// TIA Portal V20 export
FUNCTION_BLOCK "Sequence_2_JROutPnPRight"   // FB32847, LAD
TITLE = Sequence
// Sequence template programmend in ladder logic
// stored: IsIECCheckEnabled true, MemoryReserve 100, Namespace Unit1.Em2, SetENOAutomatically true
   VAR_INPUT
      unitStatus : "LAF_typeUnitStatus";
   END_VAR
   VAR
      instSequenceLADControl { ExternalWritable := 'False'} : "LAF_ControlLadSequence";
      instSequenceLADStatus { ExternalWritable := 'False'} : "LAF_StatusLadSequence";
      statTonTime { ExternalWritable := 'False'} : Array[0..9999] of TON_TIME;
      NoDataCheck { S7_SetPoint := 'True'} : "LER_typePartData";
   END_VAR
   VAR_TEMP
      tempCustomerAction : Bool;   // Placeholder for possible actions
      tempDo_nothing_and_wait_for_init : Bool;   // Placeholder for doing nothing
      tempSafeStateCondition : Bool;   // Temp Condition for the equipment module to be in a safe state
   END_VAR
   VAR CONSTANT
      FALSE : Bool := FALSE;
      delayTime : Time := T#100ms;
      STEP_IDLE : DInt := 1;
      JOB_1_STEP_01 : DInt := 101;
      JOB_1_STEP_10 : DInt := 110;
      JOB_1_STEP_20 : DInt := 120;
      JOB_1_STEP_30 : DInt := 130;
      JOB_1_STEP_40 : DInt := 140;
      JOB_1_STEP_50 : DInt := 150;
      JOB_1_STEP_60 : DInt := 160;
      JOB_1_STEP_70 : DInt := 170;
      JOB_1_STEP_80 : DInt := 180;
      JOB_1_STEP_90 : DInt := 190;
      JOB_2_STEP_1 : DInt := 201;
      JOB_2_STEP_10 : DInt := 210;
      JOB_2_STEP_11 : DInt := 211;
      JOB_2_STEP_12 : DInt := 212;
      JOB_2_STEP_20 : DInt := 220;
      JOB_2_STEP_21 : DInt := 221;
      JOB_2_STEP_22 : DInt := 222;
      JOB_2_STEP_23 : DInt := 223;
      JOB_2_STEP_24 : DInt := 224;
      JOB_2_STEP_25 : DInt := 225;
      JOB_2_STEP_26 : DInt := 226;
      JOB_2_STEP_27 : DInt := 227;
      JOB_2_STEP_30 : DInt := 230;
      JOB_2_STEP_40 : DInt := 240;
      JOB_2_STEP_50 : DInt := 250;
      JOB_2_STEP_60 : DInt := 260;
      JOB_2_STEP_70 : DInt := 270;
      JOB_2_STEP_80 : DInt := 280;
      JOB_2_STEP_90 : DInt := 290;
      JOB_3_STEP_1 : DInt := 301;
      JOB_3_STEP_10 : DInt := 310;
      JOB_3_STEP_11 : DInt := 311;
      JOB_3_STEP_12 : DInt := 312;
      JOB_3_STEP_20 : DInt := 320;
      JOB_3_STEP_21 : DInt := 321;
      JOB_3_STEP_22 : DInt := 322;
      JOB_3_STEP_23 : DInt := 323;
      JOB_3_STEP_24 : DInt := 324;
      JOB_3_STEP_25 : DInt := 325;
      JOB_3_STEP_26 : DInt := 326;
      JOB_3_STEP_27 : DInt := 327;
      JOB_3_STEP_30 : DInt := 330;
      JOB_3_STEP_42 : DInt;
      JOB_3_STEP_31 : DInt := 331;
      JOB_3_STEP_40 : DInt := 340;
      JOB_3_STEP_41 : DInt := 341;
      JOB_3_STEP_50 : DInt := 350;
      JOB_3_STEP_51 : DInt := 351;
      JOB_3_STEP_60 : DInt := 360;
      JOB_3_STEP_70 : DInt := 370;
      JOB_3_STEP_80 : DInt := 380;
      JOB_3_STEP_90 : DInt := 390;
      STEP_IMMEDIATE_STOP : DInt := 9001;   // Step executed when an immediate stop command is triggered for the sequence (i.e. when unit is in state aborting)
      TO_DO_INSERT_ACTIONS_HERE : Bool := TRUE;   // Template : Add actions
      TO_DO_INSERT_CONDITION_FOR_TRANSITION_HERE : Bool := TRUE;   // Template : Add conditions
   END_VAR
   VAR_TEMP   // added for the SCL form of the ladder/FBD networks
      _w1 : Bool;
      _w2 : Bool;
      _w3 : Bool;
      _w4 : Bool;
      _w5 : Bool;
      _w6 : Bool;
      _w7 : Bool;
      _w8 : Bool;
   END_VAR
BEGIN

REGION Network 1: BLOCK INFO HEADER
   // (company) / (C) Copyright (year)
   // ---------------------------------------------------------------------------------
   // Title:                             (Title of this block)
   // Comment/Function: (that is implemented in the block)
   // Library/Family:           (that the source is dedicated to)
   // Author:                        (department / person in charge / contact)
   // Target System:          (test system with FW version)
   // Engineering:              TIA Portal (SW version)
   // Restrictions:               (OB types, etc.)
   // Requirements:           (hardware, technological package, etc.)
   // ---------------------------------------------------------------------------------
   // Change log table:
   // Version          | Date             | Signature      | Expert in charge  | Changes applied ------------------------|----------------------|-------------------------|--------------------------------|-----------------------
   // 001.000.000 | yyyy-mm-dd | 0x00000000 | (name of expert) | First released version
END_REGION

REGION Network 2: DESCRIPTION
   // This is a template block provided by the Automation Framework. It can be used to create an own project.
   // The Block Info Header is prepared to put in your own data.
   // Description of the block could be added here and the docu created by Code2Docu.
END_REGION

REGION Network 3: *************** CONTROL **********************
END_REGION

REGION Network 4: Sequence Control ("Enter your Sequins number here")
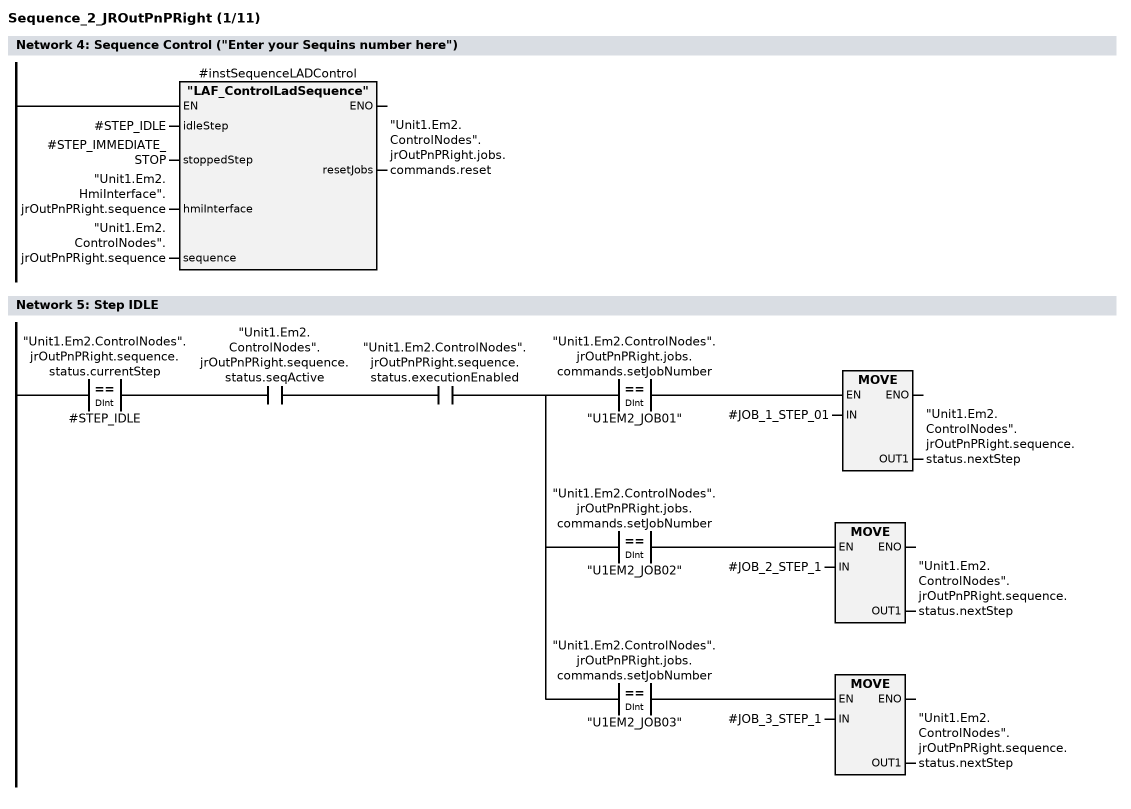
   RUNG wire#powerrail
      #instSequenceLADControl(idleStep := #STEP_IDLE, stoppedStep := #STEP_IMMEDIATE_STOP, hmiInterface := "Unit1.Em2.HmiInterface".jrOutPnPRight.sequence, sequence := "Unit1.Em2.ControlNodes".jrOutPnPRight.sequence, resetJobs => "Unit1.Em2.ControlNodes".jrOutPnPRight.jobs.commands.reset)
   END_RUNG
   // the same network as SCL:
   #instSequenceLADControl(idleStep := #STEP_IDLE,   // "LAF_ControlLadSequence"
                           stoppedStep := #STEP_IMMEDIATE_STOP,
                           hmiInterface := "Unit1.Em2.HmiInterface".jrOutPnPRight.sequence,
                           sequence := "Unit1.Em2.ControlNodes".jrOutPnPRight.sequence,
                           resetJobs => "Unit1.Em2.ControlNodes".jrOutPnPRight.jobs.commands.reset);
END_REGION

REGION Network 5: Step IDLE
   RUNG wire#powerrail
      { S7_Templates := "SrcType := DInt" } EQ_Contact(in1 := "Unit1.Em2.ControlNodes".jrOutPnPRight.sequence.status.currentStep, in2 := #STEP_IDLE)
      Contact( "Unit1.Em2.ControlNodes".jrOutPnPRight.sequence.status.seqActive )
      Contact( "Unit1.Em2.ControlNodes".jrOutPnPRight.sequence.status.executionEnabled )
      wire#w1
      { S7_Templates := "SrcType := DInt" } EQ_Contact(in1 := "Unit1.Em2.ControlNodes".jrOutPnPRight.jobs.commands.setJobNumber, in2 := "U1EM2_JOB01")
      Move(in := #JOB_1_STEP_01, out1 => "Unit1.Em2.ControlNodes".jrOutPnPRight.sequence.status.nextStep)
   END_RUNG
   RUNG wire#w1
      { S7_Templates := "SrcType := DInt" } EQ_Contact(in1 := "Unit1.Em2.ControlNodes".jrOutPnPRight.jobs.commands.setJobNumber, in2 := "U1EM2_JOB02")
      Move(in := #JOB_2_STEP_1, out1 => "Unit1.Em2.ControlNodes".jrOutPnPRight.sequence.status.nextStep)
   END_RUNG
   RUNG wire#w1
      { S7_Templates := "SrcType := DInt" } EQ_Contact(in1 := "Unit1.Em2.ControlNodes".jrOutPnPRight.jobs.commands.setJobNumber, in2 := "U1EM2_JOB03")
      Move(in := #JOB_3_STEP_1, out1 => "Unit1.Em2.ControlNodes".jrOutPnPRight.sequence.status.nextStep)
   END_RUNG
   // the same network as SCL:
   #_w1 := ("Unit1.Em2.ControlNodes".jrOutPnPRight.sequence.status.currentStep = #STEP_IDLE) AND "Unit1.Em2.ControlNodes".jrOutPnPRight.sequence.status.seqActive AND "Unit1.Em2.ControlNodes".jrOutPnPRight.sequence.status.executionEnabled;
   IF #_w1 AND ("Unit1.Em2.ControlNodes".jrOutPnPRight.jobs.commands.setJobNumber = "U1EM2_JOB01") THEN
       "Unit1.Em2.ControlNodes".jrOutPnPRight.sequence.status.nextStep := #JOB_1_STEP_01;
   END_IF;
   IF #_w1 AND ("Unit1.Em2.ControlNodes".jrOutPnPRight.jobs.commands.setJobNumber = "U1EM2_JOB02") THEN
       "Unit1.Em2.ControlNodes".jrOutPnPRight.sequence.status.nextStep := #JOB_2_STEP_1;
   END_IF;
   IF #_w1 AND ("Unit1.Em2.ControlNodes".jrOutPnPRight.jobs.commands.setJobNumber = "U1EM2_JOB03") THEN
       "Unit1.Em2.ControlNodes".jrOutPnPRight.sequence.status.nextStep := #JOB_3_STEP_1;
   END_IF;
END_REGION

REGION Network 6: *************** JOB[1] HOMING *************************
END_REGION

REGION Network 7: Step[101] : JOB[1] Condition
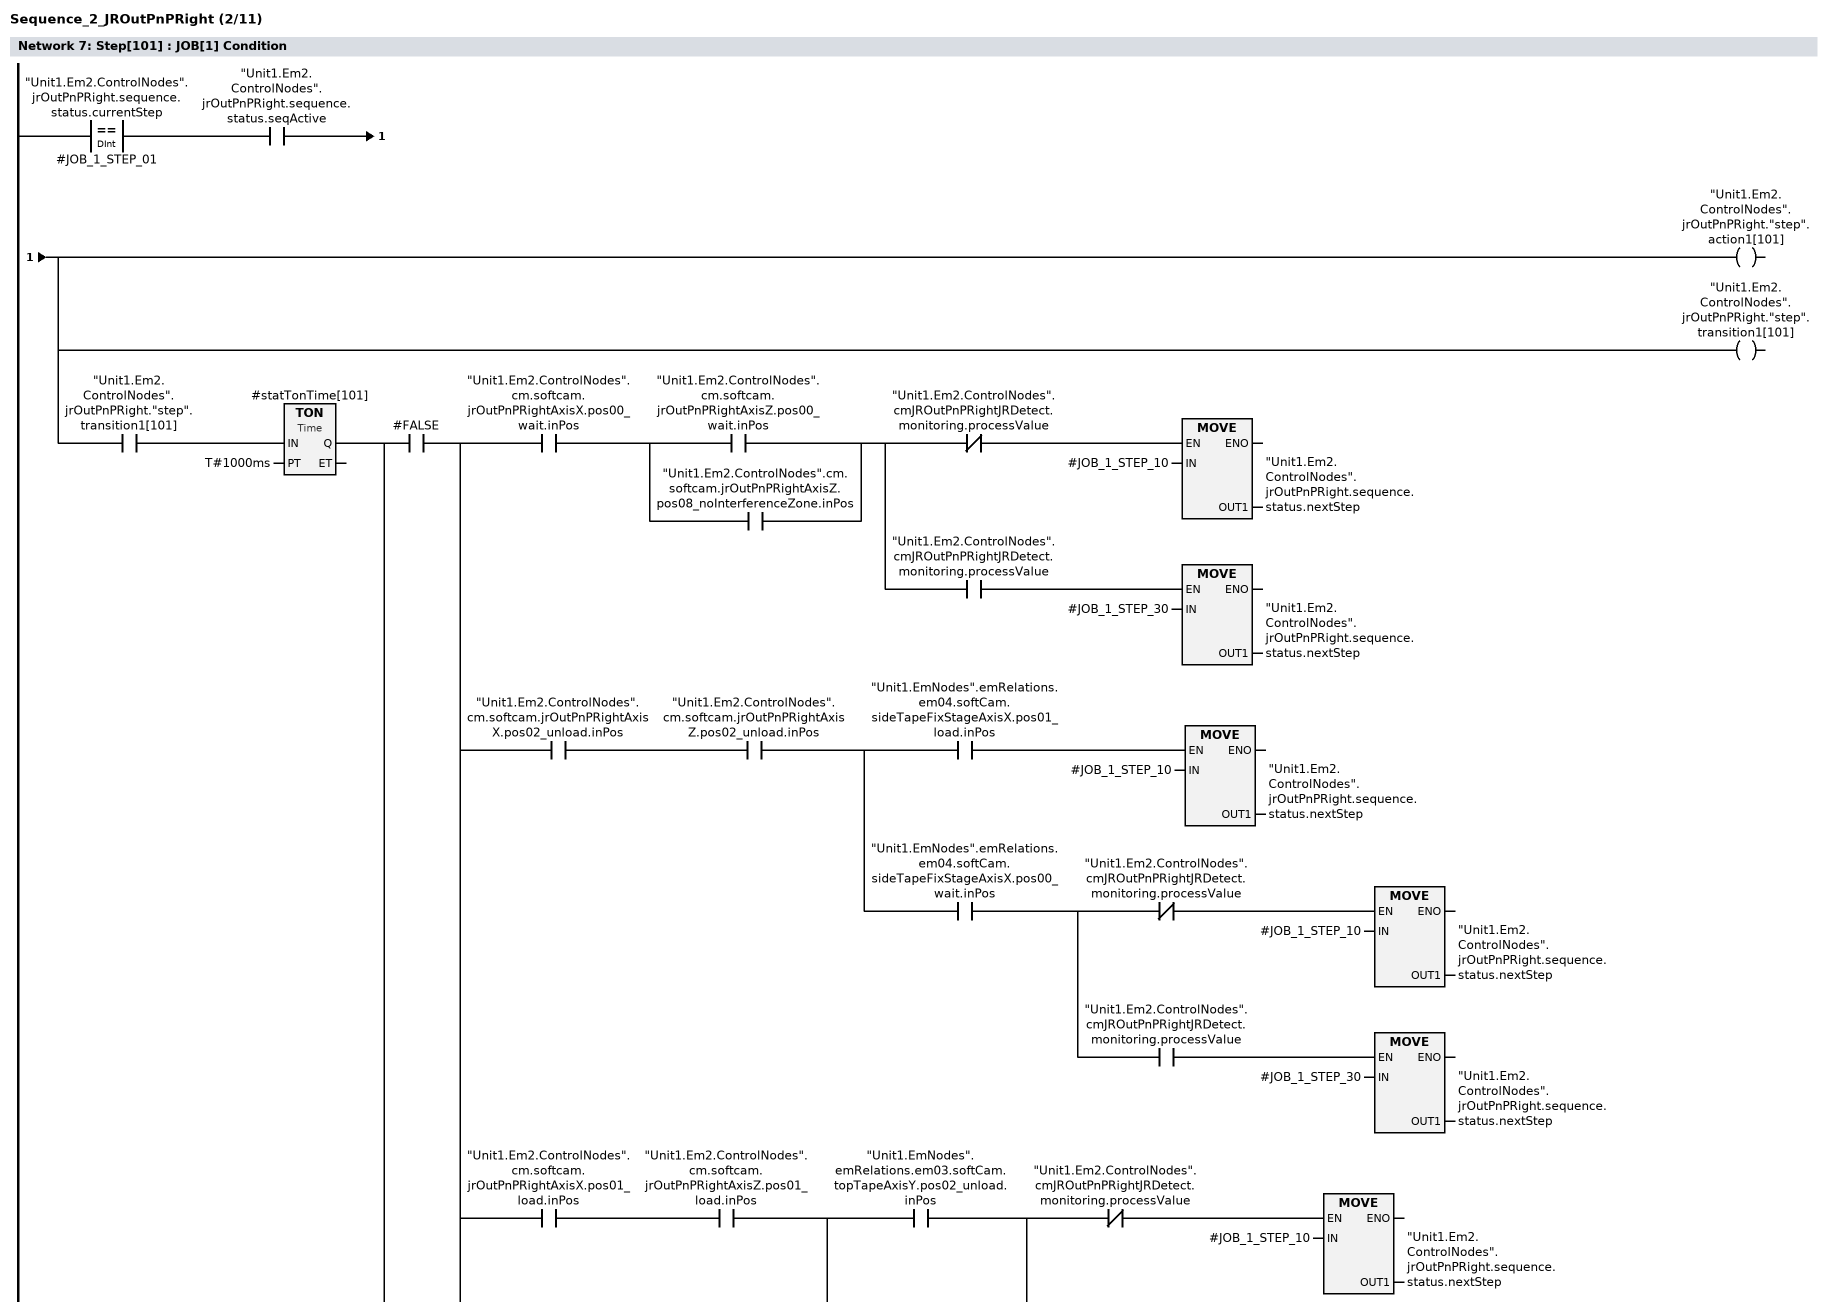
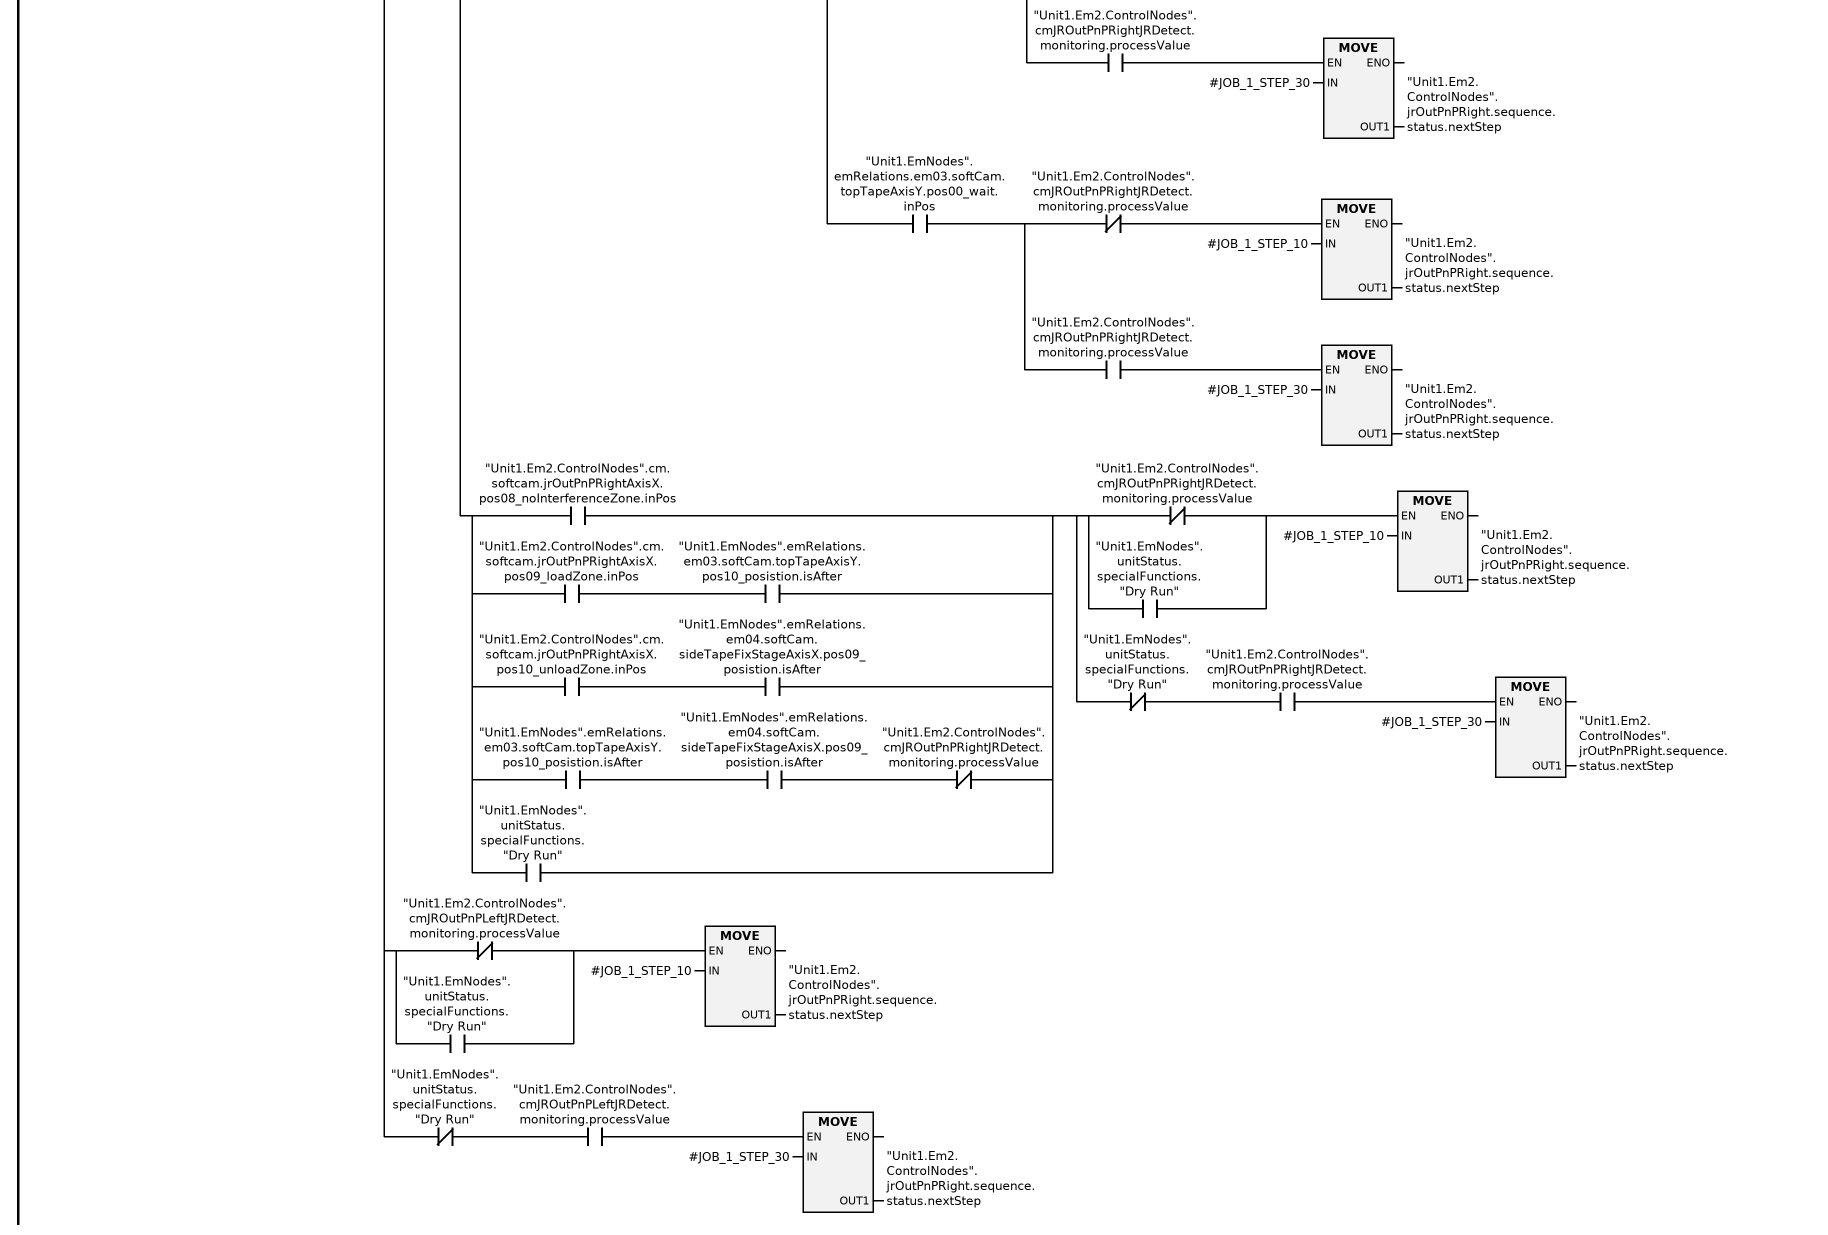
   RUNG wire#powerrail
      { S7_Templates := "SrcType := DInt" } EQ_Contact(in1 := "Unit1.Em2.ControlNodes".jrOutPnPRight.sequence.status.currentStep, in2 := #JOB_1_STEP_01)
      Contact( "Unit1.Em2.ControlNodes".jrOutPnPRight.sequence.status.seqActive )
      wire#w1
      Coil( "Unit1.Em2.ControlNodes".jrOutPnPRight."step".action1[101] )
   END_RUNG
   RUNG wire#w1
      Coil( "Unit1.Em2.ControlNodes".jrOutPnPRight."step".transition1[101] )
   END_RUNG
   RUNG wire#w1
      Contact( "Unit1.Em2.ControlNodes".jrOutPnPRight."step".transition1[101] )
      { S7_Templates := "time_type := Time" } #statTonTime[101].TON(pt := T#1000ms, et =>)
      wire#w2
      Contact( #FALSE )
      wire#w3
      Contact( "Unit1.Em2.ControlNodes".cm.softcam.jrOutPnPRightAxisX.pos00_wait.inPos )
      wire#w4
      Contact( "Unit1.Em2.ControlNodes".cm.softcam.jrOutPnPRightAxisZ.pos00_wait.inPos )
      wire#w5
      I_Contact( "Unit1.Em2.ControlNodes".cmJROutPnPRightJRDetect.monitoring.processValue )
      Move(in := #JOB_1_STEP_10, out1 => "Unit1.Em2.ControlNodes".jrOutPnPRight.sequence.status.nextStep)
   END_RUNG
   RUNG wire#w4
      Contact( "Unit1.Em2.ControlNodes".cm.softcam.jrOutPnPRightAxisZ.pos08_noInterferenceZone.inPos )
   END_RUNG wire#w5
   RUNG wire#w5
      Contact( "Unit1.Em2.ControlNodes".cmJROutPnPRightJRDetect.monitoring.processValue )
      Move(in := #JOB_1_STEP_30, out1 => "Unit1.Em2.ControlNodes".jrOutPnPRight.sequence.status.nextStep)
   END_RUNG
   RUNG wire#w3
      Contact( "Unit1.Em2.ControlNodes".cm.softcam.jrOutPnPRightAxisX.pos02_unload.inPos )
      Contact( "Unit1.Em2.ControlNodes".cm.softcam.jrOutPnPRightAxisZ.pos02_unload.inPos )
      wire#w6
      Contact( "Unit1.EmNodes".emRelations.em04.softCam.sideTapeFixStageAxisX.pos01_load.inPos )
      Move(in := #JOB_1_STEP_10, out1 => "Unit1.Em2.ControlNodes".jrOutPnPRight.sequence.status.nextStep)
   END_RUNG
   RUNG wire#w6
      Contact( "Unit1.EmNodes".emRelations.em04.softCam.sideTapeFixStageAxisX.pos00_wait.inPos )
      wire#w7
      I_Contact( "Unit1.Em2.ControlNodes".cmJROutPnPRightJRDetect.monitoring.processValue )
      Move(in := #JOB_1_STEP_10, out1 => "Unit1.Em2.ControlNodes".jrOutPnPRight.sequence.status.nextStep)
   END_RUNG
   RUNG wire#w7
      Contact( "Unit1.Em2.ControlNodes".cmJROutPnPRightJRDetect.monitoring.processValue )
      Move(in := #JOB_1_STEP_30, out1 => "Unit1.Em2.ControlNodes".jrOutPnPRight.sequence.status.nextStep)
   END_RUNG
   RUNG wire#w3
      Contact( "Unit1.Em2.ControlNodes".cm.softcam.jrOutPnPRightAxisX.pos01_load.inPos )
      Contact( "Unit1.Em2.ControlNodes".cm.softcam.jrOutPnPRightAxisZ.pos01_load.inPos )
      wire#w8
      Contact( "Unit1.EmNodes".emRelations.em03.softCam.topTapeAxisY.pos02_unload.inPos )
      wire#w9
      I_Contact( "Unit1.Em2.ControlNodes".cmJROutPnPRightJRDetect.monitoring.processValue )
      Move(in := #JOB_1_STEP_10, out1 => "Unit1.Em2.ControlNodes".jrOutPnPRight.sequence.status.nextStep)
   END_RUNG
   RUNG wire#w9
      Contact( "Unit1.Em2.ControlNodes".cmJROutPnPRightJRDetect.monitoring.processValue )
      Move(in := #JOB_1_STEP_30, out1 => "Unit1.Em2.ControlNodes".jrOutPnPRight.sequence.status.nextStep)
   END_RUNG
   RUNG wire#w8
      Contact( "Unit1.EmNodes".emRelations.em03.softCam.topTapeAxisY.pos00_wait.inPos )
      wire#w10
      I_Contact( "Unit1.Em2.ControlNodes".cmJROutPnPRightJRDetect.monitoring.processValue )
      Move(in := #JOB_1_STEP_10, out1 => "Unit1.Em2.ControlNodes".jrOutPnPRight.sequence.status.nextStep)
   END_RUNG
   RUNG wire#w10
      Contact( "Unit1.Em2.ControlNodes".cmJROutPnPRightJRDetect.monitoring.processValue )
      Move(in := #JOB_1_STEP_30, out1 => "Unit1.Em2.ControlNodes".jrOutPnPRight.sequence.status.nextStep)
   END_RUNG
   RUNG wire#w3
      Contact( "Unit1.Em2.ControlNodes".cm.softcam.jrOutPnPRightAxisX.pos08_noInterferenceZone.inPos )
      wire#w11
      I_Contact( "Unit1.Em2.ControlNodes".cmJROutPnPRightJRDetect.monitoring.processValue )
      wire#w12
      Move(in := #JOB_1_STEP_10, out1 => "Unit1.Em2.ControlNodes".jrOutPnPRight.sequence.status.nextStep)
   END_RUNG
   RUNG wire#w3
      Contact( "Unit1.Em2.ControlNodes".cm.softcam.jrOutPnPRightAxisX.pos09_loadZone.inPos )
      Contact( "Unit1.EmNodes".emRelations.em03.softCam.topTapeAxisY.pos10_posistion.isAfter )
   END_RUNG wire#w11
   RUNG wire#w3
      Contact( "Unit1.Em2.ControlNodes".cm.softcam.jrOutPnPRightAxisX.pos10_unloadZone.inPos )
      Contact( "Unit1.EmNodes".emRelations.em04.softCam.sideTapeFixStageAxisX.pos09_posistion.isAfter )
   END_RUNG wire#w11
   RUNG wire#w3
      Contact( "Unit1.EmNodes".emRelations.em03.softCam.topTapeAxisY.pos10_posistion.isAfter )
      Contact( "Unit1.EmNodes".emRelations.em04.softCam.sideTapeFixStageAxisX.pos09_posistion.isAfter )
      I_Contact( "Unit1.Em2.ControlNodes".cmJROutPnPRightJRDetect.monitoring.processValue )
   END_RUNG wire#w11
   RUNG wire#w3
      Contact( "Unit1.EmNodes".unitStatus.specialFunctions."Dry Run" )
   END_RUNG wire#w11
   RUNG wire#w11
      Contact( "Unit1.EmNodes".unitStatus.specialFunctions."Dry Run" )
   END_RUNG wire#w12
   RUNG wire#w11
      I_Contact( "Unit1.EmNodes".unitStatus.specialFunctions."Dry Run" )
      Contact( "Unit1.Em2.ControlNodes".cmJROutPnPRightJRDetect.monitoring.processValue )
      Move(in := #JOB_1_STEP_30, out1 => "Unit1.Em2.ControlNodes".jrOutPnPRight.sequence.status.nextStep)
   END_RUNG
   RUNG wire#w2
      I_Contact( "Unit1.Em2.ControlNodes".cmJROutPnPLeftJRDetect.monitoring.processValue )
      wire#w13
      Move(in := #JOB_1_STEP_10, out1 => "Unit1.Em2.ControlNodes".jrOutPnPRight.sequence.status.nextStep)
   END_RUNG
   RUNG wire#w2
      Contact( "Unit1.EmNodes".unitStatus.specialFunctions."Dry Run" )
   END_RUNG wire#w13
   RUNG wire#w2
      I_Contact( "Unit1.EmNodes".unitStatus.specialFunctions."Dry Run" )
      Contact( "Unit1.Em2.ControlNodes".cmJROutPnPLeftJRDetect.monitoring.processValue )
      Move(in := #JOB_1_STEP_30, out1 => "Unit1.Em2.ControlNodes".jrOutPnPRight.sequence.status.nextStep)
   END_RUNG
   // the same network as SCL:
   "Unit1.Em2.ControlNodes".jrOutPnPRight."step".action1[101] := ("Unit1.Em2.ControlNodes".jrOutPnPRight.sequence.status.currentStep = #JOB_1_STEP_01) AND "Unit1.Em2.ControlNodes".jrOutPnPRight.sequence.status.seqActive;
   "Unit1.Em2.ControlNodes".jrOutPnPRight."step".transition1[101] := ("Unit1.Em2.ControlNodes".jrOutPnPRight.sequence.status.currentStep = #JOB_1_STEP_01) AND "Unit1.Em2.ControlNodes".jrOutPnPRight.sequence.status.seqActive;
   #statTonTime[101].TON(IN := ("Unit1.Em2.ControlNodes".jrOutPnPRight.sequence.status.currentStep = #JOB_1_STEP_01) AND "Unit1.Em2.ControlNodes".jrOutPnPRight.sequence.status.seqActive AND "Unit1.Em2.ControlNodes".jrOutPnPRight."step".transition1[101],
                         PT := T#1000ms);
   #_w1 := #statTonTime[101].Q AND #FALSE;
   #_w2 := #_w1 AND "Unit1.Em2.ControlNodes".cm.softcam.jrOutPnPRightAxisX.pos00_wait.inPos AND ("Unit1.Em2.ControlNodes".cm.softcam.jrOutPnPRightAxisZ.pos00_wait.inPos OR "Unit1.Em2.ControlNodes".cm.softcam.jrOutPnPRightAxisZ.pos08_noInterferenceZone.inPos);
   IF #_w2 AND NOT "Unit1.Em2.ControlNodes".cmJROutPnPRightJRDetect.monitoring.processValue THEN
       "Unit1.Em2.ControlNodes".jrOutPnPRight.sequence.status.nextStep := #JOB_1_STEP_10;
   END_IF;
   IF #_w2 AND "Unit1.Em2.ControlNodes".cmJROutPnPRightJRDetect.monitoring.processValue THEN
       "Unit1.Em2.ControlNodes".jrOutPnPRight.sequence.status.nextStep := #JOB_1_STEP_30;
   END_IF;
   #_w3 := #_w1 AND "Unit1.Em2.ControlNodes".cm.softcam.jrOutPnPRightAxisX.pos02_unload.inPos AND "Unit1.Em2.ControlNodes".cm.softcam.jrOutPnPRightAxisZ.pos02_unload.inPos;
   IF #_w3 AND "Unit1.EmNodes".emRelations.em04.softCam.sideTapeFixStageAxisX.pos01_load.inPos THEN
       "Unit1.Em2.ControlNodes".jrOutPnPRight.sequence.status.nextStep := #JOB_1_STEP_10;
   END_IF;
   #_w4 := #_w3 AND "Unit1.EmNodes".emRelations.em04.softCam.sideTapeFixStageAxisX.pos00_wait.inPos;
   IF #_w4 AND NOT "Unit1.Em2.ControlNodes".cmJROutPnPRightJRDetect.monitoring.processValue THEN
       "Unit1.Em2.ControlNodes".jrOutPnPRight.sequence.status.nextStep := #JOB_1_STEP_10;
   END_IF;
   IF #_w4 AND "Unit1.Em2.ControlNodes".cmJROutPnPRightJRDetect.monitoring.processValue THEN
       "Unit1.Em2.ControlNodes".jrOutPnPRight.sequence.status.nextStep := #JOB_1_STEP_30;
   END_IF;
   #_w5 := #_w1 AND "Unit1.Em2.ControlNodes".cm.softcam.jrOutPnPRightAxisX.pos01_load.inPos AND "Unit1.Em2.ControlNodes".cm.softcam.jrOutPnPRightAxisZ.pos01_load.inPos;
   #_w6 := #_w5 AND "Unit1.EmNodes".emRelations.em03.softCam.topTapeAxisY.pos02_unload.inPos;
   IF #_w6 AND NOT "Unit1.Em2.ControlNodes".cmJROutPnPRightJRDetect.monitoring.processValue THEN
       "Unit1.Em2.ControlNodes".jrOutPnPRight.sequence.status.nextStep := #JOB_1_STEP_10;
   END_IF;
   IF #_w6 AND "Unit1.Em2.ControlNodes".cmJROutPnPRightJRDetect.monitoring.processValue THEN
       "Unit1.Em2.ControlNodes".jrOutPnPRight.sequence.status.nextStep := #JOB_1_STEP_30;
   END_IF;
   #_w7 := #_w5 AND "Unit1.EmNodes".emRelations.em03.softCam.topTapeAxisY.pos00_wait.inPos;
   IF #_w7 AND NOT "Unit1.Em2.ControlNodes".cmJROutPnPRightJRDetect.monitoring.processValue THEN
       "Unit1.Em2.ControlNodes".jrOutPnPRight.sequence.status.nextStep := #JOB_1_STEP_10;
   END_IF;
   IF #_w7 AND "Unit1.Em2.ControlNodes".cmJROutPnPRightJRDetect.monitoring.processValue THEN
       "Unit1.Em2.ControlNodes".jrOutPnPRight.sequence.status.nextStep := #JOB_1_STEP_30;
   END_IF;
   #_w8 := #_w1 AND ("Unit1.Em2.ControlNodes".cm.softcam.jrOutPnPRightAxisX.pos08_noInterferenceZone.inPos OR ("Unit1.Em2.ControlNodes".cm.softcam.jrOutPnPRightAxisX.pos09_loadZone.inPos AND "Unit1.EmNodes".emRelations.em03.softCam.topTapeAxisY.pos10_posistion.isAfter) OR ("Unit1.Em2.ControlNodes".cm.softcam.jrOutPnPRightAxisX.pos10_unloadZone.inPos AND "Unit1.EmNodes".emRelations.em04.softCam.sideTapeFixStageAxisX.pos09_posistion.isAfter) OR ("Unit1.EmNodes".emRelations.em03.softCam.topTapeAxisY.pos10_posistion.isAfter AND "Unit1.EmNodes".emRelations.em04.softCam.sideTapeFixStageAxisX.pos09_posistion.isAfter AND NOT "Unit1.Em2.ControlNodes".cmJROutPnPRightJRDetect.monitoring.processValue) OR "Unit1.EmNodes".unitStatus.specialFunctions."Dry Run");
   IF #_w8 AND (NOT "Unit1.Em2.ControlNodes".cmJROutPnPRightJRDetect.monitoring.processValue OR "Unit1.EmNodes".unitStatus.specialFunctions."Dry Run") THEN
       "Unit1.Em2.ControlNodes".jrOutPnPRight.sequence.status.nextStep := #JOB_1_STEP_10;
   END_IF;
   IF #_w8 AND NOT "Unit1.EmNodes".unitStatus.specialFunctions."Dry Run" AND "Unit1.Em2.ControlNodes".cmJROutPnPRightJRDetect.monitoring.processValue THEN
       "Unit1.Em2.ControlNodes".jrOutPnPRight.sequence.status.nextStep := #JOB_1_STEP_30;
   END_IF;
   IF #statTonTime[101].Q AND (NOT "Unit1.Em2.ControlNodes".cmJROutPnPLeftJRDetect.monitoring.processValue OR "Unit1.EmNodes".unitStatus.specialFunctions."Dry Run") THEN
       "Unit1.Em2.ControlNodes".jrOutPnPRight.sequence.status.nextStep := #JOB_1_STEP_10;
   END_IF;
   IF #statTonTime[101].Q AND NOT "Unit1.EmNodes".unitStatus.specialFunctions."Dry Run" AND "Unit1.Em2.ControlNodes".cmJROutPnPLeftJRDetect.monitoring.processValue THEN
       "Unit1.Em2.ControlNodes".jrOutPnPRight.sequence.status.nextStep := #JOB_1_STEP_30;
   END_IF;
END_REGION

REGION Network 8: Step[110] : JR PP Right Clamp Open
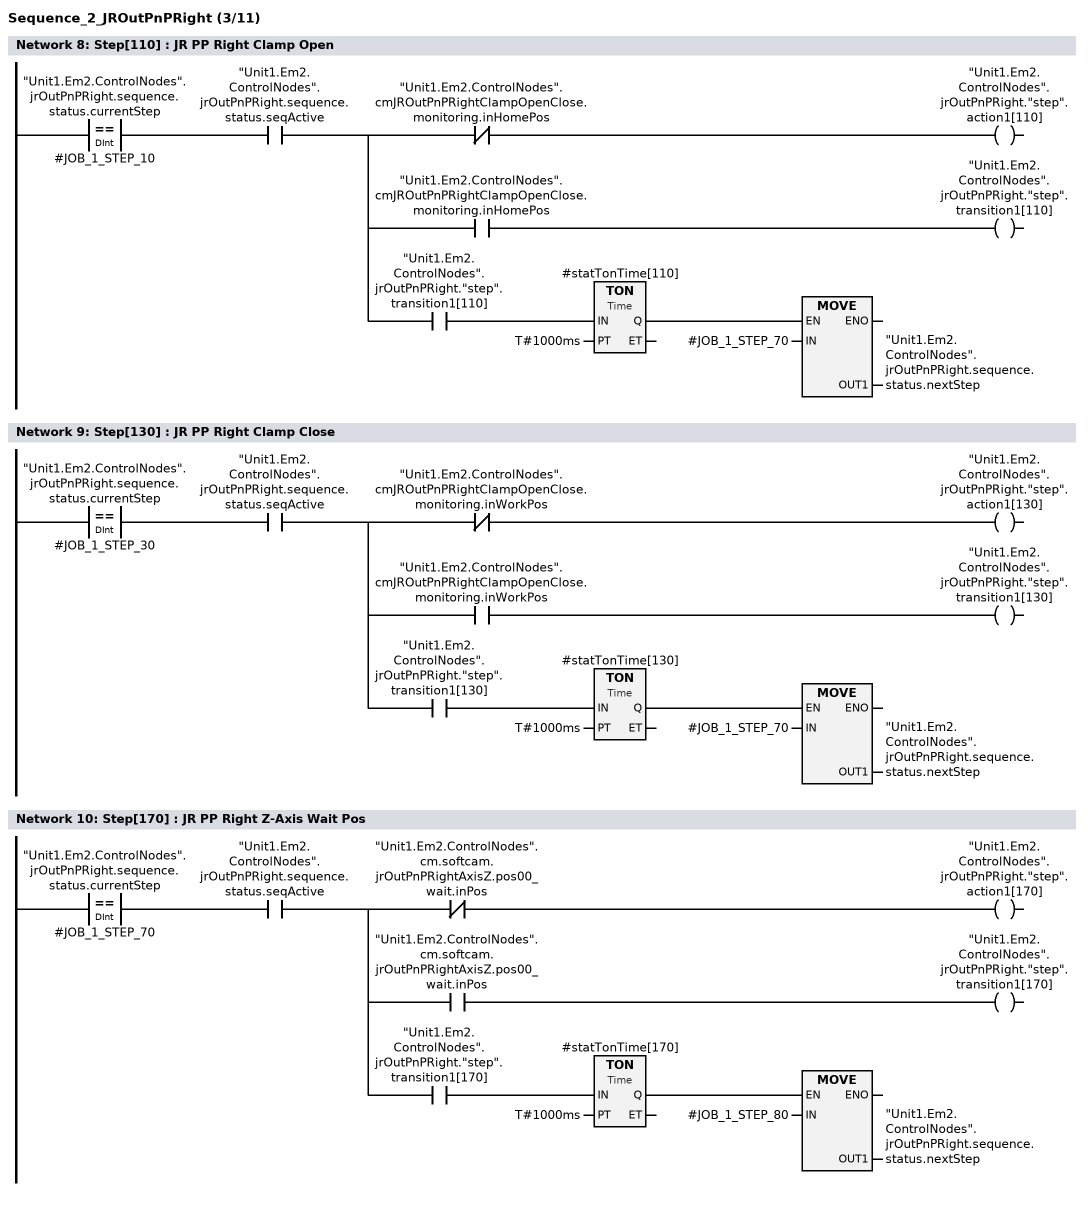
   RUNG wire#powerrail
      { S7_Templates := "SrcType := DInt" } EQ_Contact(in1 := "Unit1.Em2.ControlNodes".jrOutPnPRight.sequence.status.currentStep, in2 := #JOB_1_STEP_10)
      Contact( "Unit1.Em2.ControlNodes".jrOutPnPRight.sequence.status.seqActive )
      wire#w1
      I_Contact( "Unit1.Em2.ControlNodes".cmJROutPnPRightClampOpenClose.monitoring.inHomePos )
      Coil( "Unit1.Em2.ControlNodes".jrOutPnPRight."step".action1[110] )
   END_RUNG
   RUNG wire#w1
      Contact( "Unit1.Em2.ControlNodes".cmJROutPnPRightClampOpenClose.monitoring.inHomePos )
      Coil( "Unit1.Em2.ControlNodes".jrOutPnPRight."step".transition1[110] )
   END_RUNG
   RUNG wire#w1
      Contact( "Unit1.Em2.ControlNodes".jrOutPnPRight."step".transition1[110] )
      { S7_Templates := "time_type := Time" } #statTonTime[110].TON(pt := T#1000ms, et =>)
      Move(in := #JOB_1_STEP_70, out1 => "Unit1.Em2.ControlNodes".jrOutPnPRight.sequence.status.nextStep)
   END_RUNG
   // the same network as SCL:
   #_w1 := ("Unit1.Em2.ControlNodes".jrOutPnPRight.sequence.status.currentStep = #JOB_1_STEP_10) AND "Unit1.Em2.ControlNodes".jrOutPnPRight.sequence.status.seqActive;
   "Unit1.Em2.ControlNodes".jrOutPnPRight."step".action1[110] := #_w1 AND NOT "Unit1.Em2.ControlNodes".cmJROutPnPRightClampOpenClose.monitoring.inHomePos;
   "Unit1.Em2.ControlNodes".jrOutPnPRight."step".transition1[110] := #_w1 AND "Unit1.Em2.ControlNodes".cmJROutPnPRightClampOpenClose.monitoring.inHomePos;
   #statTonTime[110].TON(IN := #_w1 AND "Unit1.Em2.ControlNodes".jrOutPnPRight."step".transition1[110],
                         PT := T#1000ms);
   IF #statTonTime[110].Q THEN
       "Unit1.Em2.ControlNodes".jrOutPnPRight.sequence.status.nextStep := #JOB_1_STEP_70;
   END_IF;
END_REGION

REGION Network 9: Step[130] : JR PP Right Clamp Close
   RUNG wire#powerrail
      { S7_Templates := "SrcType := DInt" } EQ_Contact(in1 := "Unit1.Em2.ControlNodes".jrOutPnPRight.sequence.status.currentStep, in2 := #JOB_1_STEP_30)
      Contact( "Unit1.Em2.ControlNodes".jrOutPnPRight.sequence.status.seqActive )
      wire#w1
      I_Contact( "Unit1.Em2.ControlNodes".cmJROutPnPRightClampOpenClose.monitoring.inWorkPos )
      Coil( "Unit1.Em2.ControlNodes".jrOutPnPRight."step".action1[130] )
   END_RUNG
   RUNG wire#w1
      Contact( "Unit1.Em2.ControlNodes".cmJROutPnPRightClampOpenClose.monitoring.inWorkPos )
      Coil( "Unit1.Em2.ControlNodes".jrOutPnPRight."step".transition1[130] )
   END_RUNG
   RUNG wire#w1
      Contact( "Unit1.Em2.ControlNodes".jrOutPnPRight."step".transition1[130] )
      { S7_Templates := "time_type := Time" } #statTonTime[130].TON(pt := T#1000ms, et =>)
      Move(in := #JOB_1_STEP_70, out1 => "Unit1.Em2.ControlNodes".jrOutPnPRight.sequence.status.nextStep)
   END_RUNG
   // the same network as SCL:
   #_w1 := ("Unit1.Em2.ControlNodes".jrOutPnPRight.sequence.status.currentStep = #JOB_1_STEP_30) AND "Unit1.Em2.ControlNodes".jrOutPnPRight.sequence.status.seqActive;
   "Unit1.Em2.ControlNodes".jrOutPnPRight."step".action1[130] := #_w1 AND NOT "Unit1.Em2.ControlNodes".cmJROutPnPRightClampOpenClose.monitoring.inWorkPos;
   "Unit1.Em2.ControlNodes".jrOutPnPRight."step".transition1[130] := #_w1 AND "Unit1.Em2.ControlNodes".cmJROutPnPRightClampOpenClose.monitoring.inWorkPos;
   #statTonTime[130].TON(IN := #_w1 AND "Unit1.Em2.ControlNodes".jrOutPnPRight."step".transition1[130],
                         PT := T#1000ms);
   IF #statTonTime[130].Q THEN
       "Unit1.Em2.ControlNodes".jrOutPnPRight.sequence.status.nextStep := #JOB_1_STEP_70;
   END_IF;
END_REGION

REGION Network 10: Step[170] : JR PP Right Z-Axis Wait Pos
   RUNG wire#powerrail
      { S7_Templates := "SrcType := DInt" } EQ_Contact(in1 := "Unit1.Em2.ControlNodes".jrOutPnPRight.sequence.status.currentStep, in2 := #JOB_1_STEP_70)
      Contact( "Unit1.Em2.ControlNodes".jrOutPnPRight.sequence.status.seqActive )
      wire#w1
      I_Contact( "Unit1.Em2.ControlNodes".cm.softcam.jrOutPnPRightAxisZ.pos00_wait.inPos )
      Coil( "Unit1.Em2.ControlNodes".jrOutPnPRight."step".action1[170] )
   END_RUNG
   RUNG wire#w1
      Contact( "Unit1.Em2.ControlNodes".cm.softcam.jrOutPnPRightAxisZ.pos00_wait.inPos )
      Coil( "Unit1.Em2.ControlNodes".jrOutPnPRight."step".transition1[170] )
   END_RUNG
   RUNG wire#w1
      Contact( "Unit1.Em2.ControlNodes".jrOutPnPRight."step".transition1[170] )
      { S7_Templates := "time_type := Time" } #statTonTime[170].TON(pt := T#1000ms, et =>)
      Move(in := #JOB_1_STEP_80, out1 => "Unit1.Em2.ControlNodes".jrOutPnPRight.sequence.status.nextStep)
   END_RUNG
   // the same network as SCL:
   #_w1 := ("Unit1.Em2.ControlNodes".jrOutPnPRight.sequence.status.currentStep = #JOB_1_STEP_70) AND "Unit1.Em2.ControlNodes".jrOutPnPRight.sequence.status.seqActive;
   "Unit1.Em2.ControlNodes".jrOutPnPRight."step".action1[170] := #_w1 AND NOT "Unit1.Em2.ControlNodes".cm.softcam.jrOutPnPRightAxisZ.pos00_wait.inPos;
   "Unit1.Em2.ControlNodes".jrOutPnPRight."step".transition1[170] := #_w1 AND "Unit1.Em2.ControlNodes".cm.softcam.jrOutPnPRightAxisZ.pos00_wait.inPos;
   #statTonTime[170].TON(IN := #_w1 AND "Unit1.Em2.ControlNodes".jrOutPnPRight."step".transition1[170],
                         PT := T#1000ms);
   IF #statTonTime[170].Q THEN
       "Unit1.Em2.ControlNodes".jrOutPnPRight.sequence.status.nextStep := #JOB_1_STEP_80;
   END_IF;
END_REGION

REGION Network 11: Step[180] : JR PP Right X-Axis Wait Pos
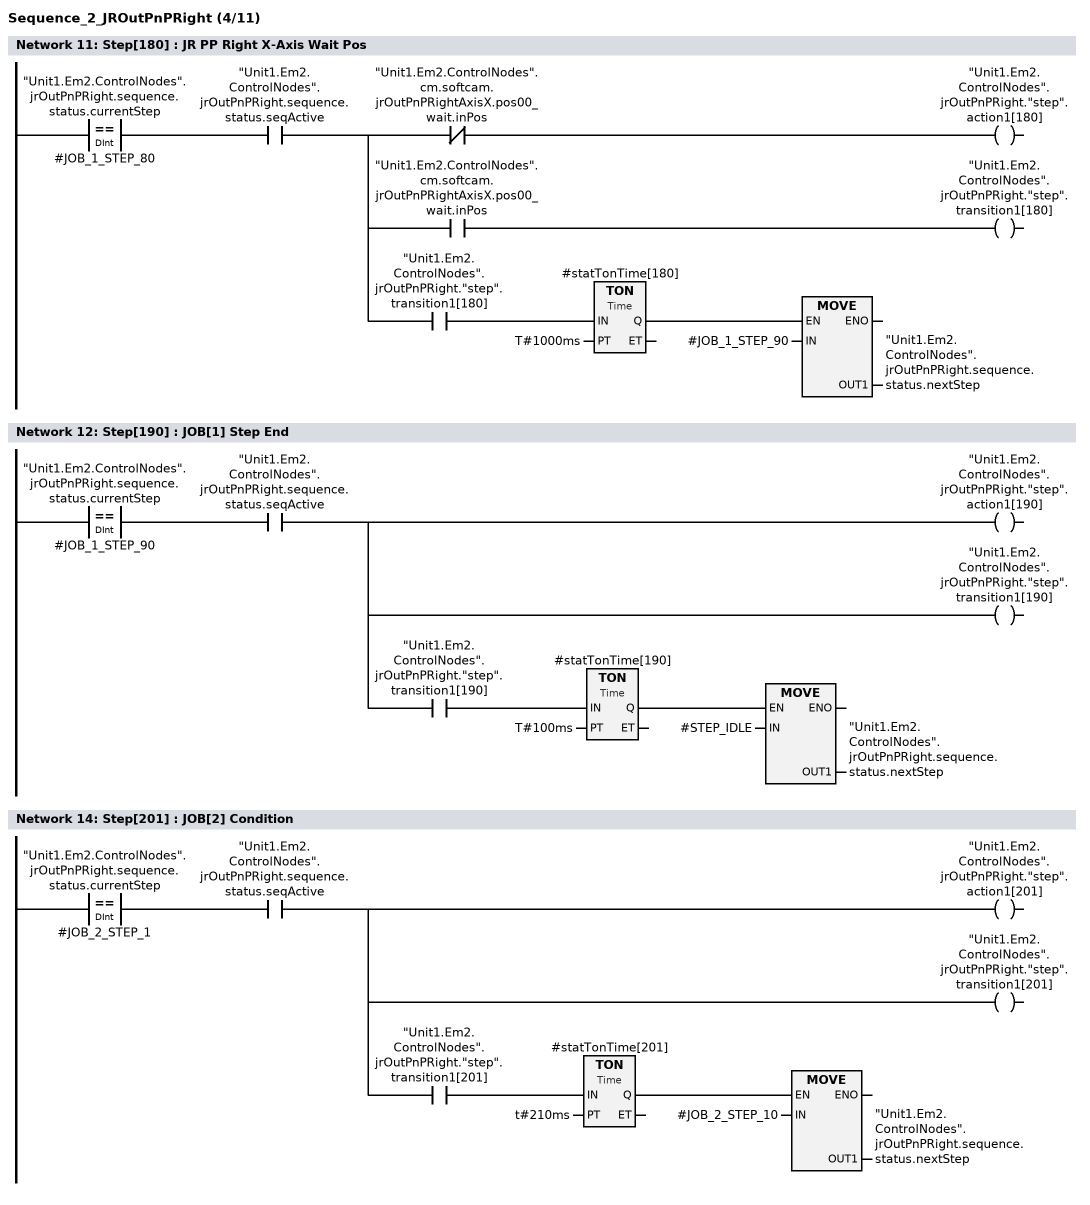
   RUNG wire#powerrail
      { S7_Templates := "SrcType := DInt" } EQ_Contact(in1 := "Unit1.Em2.ControlNodes".jrOutPnPRight.sequence.status.currentStep, in2 := #JOB_1_STEP_80)
      Contact( "Unit1.Em2.ControlNodes".jrOutPnPRight.sequence.status.seqActive )
      wire#w1
      I_Contact( "Unit1.Em2.ControlNodes".cm.softcam.jrOutPnPRightAxisX.pos00_wait.inPos )
      Coil( "Unit1.Em2.ControlNodes".jrOutPnPRight."step".action1[180] )
   END_RUNG
   RUNG wire#w1
      Contact( "Unit1.Em2.ControlNodes".cm.softcam.jrOutPnPRightAxisX.pos00_wait.inPos )
      Coil( "Unit1.Em2.ControlNodes".jrOutPnPRight."step".transition1[180] )
   END_RUNG
   RUNG wire#w1
      Contact( "Unit1.Em2.ControlNodes".jrOutPnPRight."step".transition1[180] )
      { S7_Templates := "time_type := Time" } #statTonTime[180].TON(pt := T#1000ms, et =>)
      Move(in := #JOB_1_STEP_90, out1 => "Unit1.Em2.ControlNodes".jrOutPnPRight.sequence.status.nextStep)
   END_RUNG
   // the same network as SCL:
   #_w1 := ("Unit1.Em2.ControlNodes".jrOutPnPRight.sequence.status.currentStep = #JOB_1_STEP_80) AND "Unit1.Em2.ControlNodes".jrOutPnPRight.sequence.status.seqActive;
   "Unit1.Em2.ControlNodes".jrOutPnPRight."step".action1[180] := #_w1 AND NOT "Unit1.Em2.ControlNodes".cm.softcam.jrOutPnPRightAxisX.pos00_wait.inPos;
   "Unit1.Em2.ControlNodes".jrOutPnPRight."step".transition1[180] := #_w1 AND "Unit1.Em2.ControlNodes".cm.softcam.jrOutPnPRightAxisX.pos00_wait.inPos;
   #statTonTime[180].TON(IN := #_w1 AND "Unit1.Em2.ControlNodes".jrOutPnPRight."step".transition1[180],
                         PT := T#1000ms);
   IF #statTonTime[180].Q THEN
       "Unit1.Em2.ControlNodes".jrOutPnPRight.sequence.status.nextStep := #JOB_1_STEP_90;
   END_IF;
END_REGION

REGION Network 12: Step[190] : JOB[1] Step End
   RUNG wire#powerrail
      { S7_Templates := "SrcType := DInt" } EQ_Contact(in1 := "Unit1.Em2.ControlNodes".jrOutPnPRight.sequence.status.currentStep, in2 := #JOB_1_STEP_90)
      Contact( "Unit1.Em2.ControlNodes".jrOutPnPRight.sequence.status.seqActive )
      wire#w1
      Coil( "Unit1.Em2.ControlNodes".jrOutPnPRight."step".action1[190] )
   END_RUNG
   RUNG wire#w1
      Coil( "Unit1.Em2.ControlNodes".jrOutPnPRight."step".transition1[190] )
   END_RUNG
   RUNG wire#w1
      Contact( "Unit1.Em2.ControlNodes".jrOutPnPRight."step".transition1[190] )
      { S7_Templates := "time_type := Time" } #statTonTime[190].TON(pt := T#100ms, et =>)
      Move(in := #STEP_IDLE, out1 => "Unit1.Em2.ControlNodes".jrOutPnPRight.sequence.status.nextStep)
   END_RUNG
   // the same network as SCL:
   "Unit1.Em2.ControlNodes".jrOutPnPRight."step".action1[190] := ("Unit1.Em2.ControlNodes".jrOutPnPRight.sequence.status.currentStep = #JOB_1_STEP_90) AND "Unit1.Em2.ControlNodes".jrOutPnPRight.sequence.status.seqActive;
   "Unit1.Em2.ControlNodes".jrOutPnPRight."step".transition1[190] := ("Unit1.Em2.ControlNodes".jrOutPnPRight.sequence.status.currentStep = #JOB_1_STEP_90) AND "Unit1.Em2.ControlNodes".jrOutPnPRight.sequence.status.seqActive;
   #statTonTime[190].TON(IN := ("Unit1.Em2.ControlNodes".jrOutPnPRight.sequence.status.currentStep = #JOB_1_STEP_90) AND "Unit1.Em2.ControlNodes".jrOutPnPRight.sequence.status.seqActive AND "Unit1.Em2.ControlNodes".jrOutPnPRight."step".transition1[190],
                         PT := T#100ms);
   IF #statTonTime[190].Q THEN
       "Unit1.Em2.ControlNodes".jrOutPnPRight.sequence.status.nextStep := #STEP_IDLE;
   END_IF;
END_REGION

REGION Network 13: *************** JOB[2] JR GET TOP TAPE FIX STAGE=AUTO *************************
END_REGION

REGION Network 14: Step[201] : JOB[2] Condition
   RUNG wire#powerrail
      { S7_Templates := "SrcType := DInt" } EQ_Contact(in1 := "Unit1.Em2.ControlNodes".jrOutPnPRight.sequence.status.currentStep, in2 := #JOB_2_STEP_1)
      Contact( "Unit1.Em2.ControlNodes".jrOutPnPRight.sequence.status.seqActive )
      wire#w1
      Coil( "Unit1.Em2.ControlNodes".jrOutPnPRight."step".action1[201] )
   END_RUNG
   RUNG wire#w1
      Coil( "Unit1.Em2.ControlNodes".jrOutPnPRight."step".transition1[201] )
   END_RUNG
   RUNG wire#w1
      Contact( "Unit1.Em2.ControlNodes".jrOutPnPRight."step".transition1[201] )
      { S7_Templates := "time_type := Time" } #statTonTime[201].TON(pt := t#210ms, et =>)
      Move(in := #JOB_2_STEP_10, out1 => "Unit1.Em2.ControlNodes".jrOutPnPRight.sequence.status.nextStep)
   END_RUNG
   // the same network as SCL:
   "Unit1.Em2.ControlNodes".jrOutPnPRight."step".action1[201] := ("Unit1.Em2.ControlNodes".jrOutPnPRight.sequence.status.currentStep = #JOB_2_STEP_1) AND "Unit1.Em2.ControlNodes".jrOutPnPRight.sequence.status.seqActive;
   "Unit1.Em2.ControlNodes".jrOutPnPRight."step".transition1[201] := ("Unit1.Em2.ControlNodes".jrOutPnPRight.sequence.status.currentStep = #JOB_2_STEP_1) AND "Unit1.Em2.ControlNodes".jrOutPnPRight.sequence.status.seqActive;
   #statTonTime[201].TON(IN := ("Unit1.Em2.ControlNodes".jrOutPnPRight.sequence.status.currentStep = #JOB_2_STEP_1) AND "Unit1.Em2.ControlNodes".jrOutPnPRight.sequence.status.seqActive AND "Unit1.Em2.ControlNodes".jrOutPnPRight."step".transition1[201],
                         PT := t#210ms);
   IF #statTonTime[201].Q THEN
       "Unit1.Em2.ControlNodes".jrOutPnPRight.sequence.status.nextStep := #JOB_2_STEP_10;
   END_IF;
END_REGION

REGION Network 15: Step[210] : JR PP Right X-Axis Loading Pos[Top Tape Fix Stage]
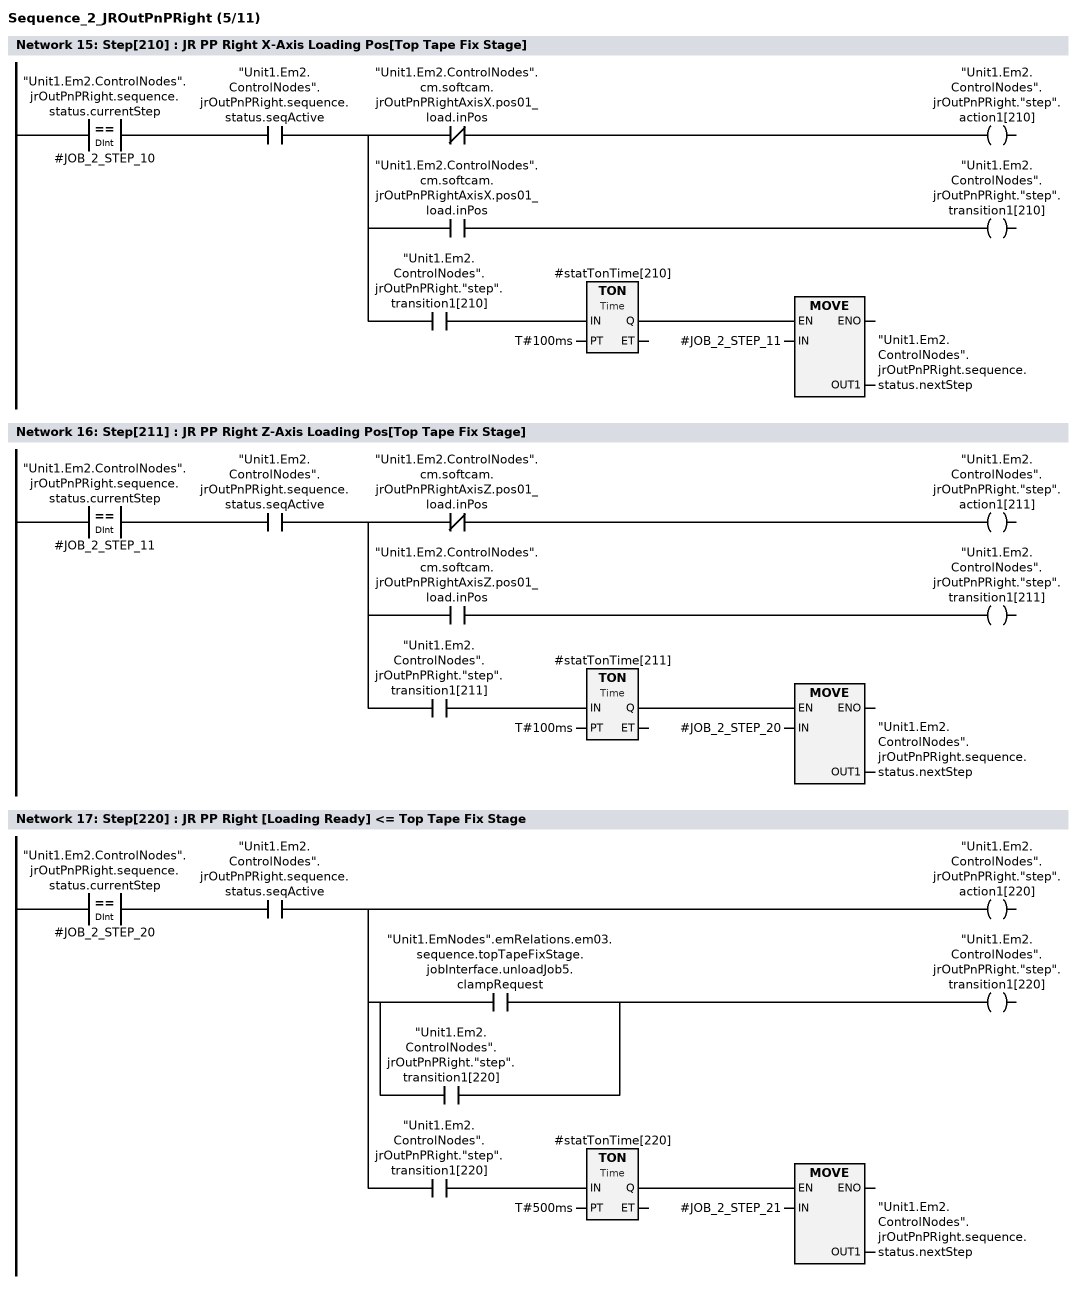
   RUNG wire#powerrail
      { S7_Templates := "SrcType := DInt" } EQ_Contact(in1 := "Unit1.Em2.ControlNodes".jrOutPnPRight.sequence.status.currentStep, in2 := #JOB_2_STEP_10)
      Contact( "Unit1.Em2.ControlNodes".jrOutPnPRight.sequence.status.seqActive )
      wire#w1
      I_Contact( "Unit1.Em2.ControlNodes".cm.softcam.jrOutPnPRightAxisX.pos01_load.inPos )
      Coil( "Unit1.Em2.ControlNodes".jrOutPnPRight."step".action1[210] )
   END_RUNG
   RUNG wire#w1
      Contact( "Unit1.Em2.ControlNodes".cm.softcam.jrOutPnPRightAxisX.pos01_load.inPos )
      Coil( "Unit1.Em2.ControlNodes".jrOutPnPRight."step".transition1[210] )
   END_RUNG
   RUNG wire#w1
      Contact( "Unit1.Em2.ControlNodes".jrOutPnPRight."step".transition1[210] )
      { S7_Templates := "time_type := Time" } #statTonTime[210].TON(pt := T#100ms, et =>)
      Move(in := #JOB_2_STEP_11, out1 => "Unit1.Em2.ControlNodes".jrOutPnPRight.sequence.status.nextStep)
   END_RUNG
   // the same network as SCL:
   #_w1 := ("Unit1.Em2.ControlNodes".jrOutPnPRight.sequence.status.currentStep = #JOB_2_STEP_10) AND "Unit1.Em2.ControlNodes".jrOutPnPRight.sequence.status.seqActive;
   "Unit1.Em2.ControlNodes".jrOutPnPRight."step".action1[210] := #_w1 AND NOT "Unit1.Em2.ControlNodes".cm.softcam.jrOutPnPRightAxisX.pos01_load.inPos;
   "Unit1.Em2.ControlNodes".jrOutPnPRight."step".transition1[210] := #_w1 AND "Unit1.Em2.ControlNodes".cm.softcam.jrOutPnPRightAxisX.pos01_load.inPos;
   #statTonTime[210].TON(IN := #_w1 AND "Unit1.Em2.ControlNodes".jrOutPnPRight."step".transition1[210],
                         PT := T#100ms);
   IF #statTonTime[210].Q THEN
       "Unit1.Em2.ControlNodes".jrOutPnPRight.sequence.status.nextStep := #JOB_2_STEP_11;
   END_IF;
END_REGION

REGION Network 16: Step[211] : JR PP Right Z-Axis Loading Pos[Top Tape Fix Stage]
   RUNG wire#powerrail
      { S7_Templates := "SrcType := DInt" } EQ_Contact(in1 := "Unit1.Em2.ControlNodes".jrOutPnPRight.sequence.status.currentStep, in2 := #JOB_2_STEP_11)
      Contact( "Unit1.Em2.ControlNodes".jrOutPnPRight.sequence.status.seqActive )
      wire#w1
      I_Contact( "Unit1.Em2.ControlNodes".cm.softcam.jrOutPnPRightAxisZ.pos01_load.inPos )
      Coil( "Unit1.Em2.ControlNodes".jrOutPnPRight."step".action1[211] )
   END_RUNG
   RUNG wire#w1
      Contact( "Unit1.Em2.ControlNodes".cm.softcam.jrOutPnPRightAxisZ.pos01_load.inPos )
      Coil( "Unit1.Em2.ControlNodes".jrOutPnPRight."step".transition1[211] )
   END_RUNG
   RUNG wire#w1
      Contact( "Unit1.Em2.ControlNodes".jrOutPnPRight."step".transition1[211] )
      { S7_Templates := "time_type := Time" } #statTonTime[211].TON(pt := T#100ms, et =>)
      Move(in := #JOB_2_STEP_20, out1 => "Unit1.Em2.ControlNodes".jrOutPnPRight.sequence.status.nextStep)
   END_RUNG
   // the same network as SCL:
   #_w1 := ("Unit1.Em2.ControlNodes".jrOutPnPRight.sequence.status.currentStep = #JOB_2_STEP_11) AND "Unit1.Em2.ControlNodes".jrOutPnPRight.sequence.status.seqActive;
   "Unit1.Em2.ControlNodes".jrOutPnPRight."step".action1[211] := #_w1 AND NOT "Unit1.Em2.ControlNodes".cm.softcam.jrOutPnPRightAxisZ.pos01_load.inPos;
   "Unit1.Em2.ControlNodes".jrOutPnPRight."step".transition1[211] := #_w1 AND "Unit1.Em2.ControlNodes".cm.softcam.jrOutPnPRightAxisZ.pos01_load.inPos;
   #statTonTime[211].TON(IN := #_w1 AND "Unit1.Em2.ControlNodes".jrOutPnPRight."step".transition1[211],
                         PT := T#100ms);
   IF #statTonTime[211].Q THEN
       "Unit1.Em2.ControlNodes".jrOutPnPRight.sequence.status.nextStep := #JOB_2_STEP_20;
   END_IF;
END_REGION

REGION Network 17: Step[220] : JR PP Right [Loading Ready] <= Top Tape Fix Stage
   RUNG wire#powerrail
      { S7_Templates := "SrcType := DInt" } EQ_Contact(in1 := "Unit1.Em2.ControlNodes".jrOutPnPRight.sequence.status.currentStep, in2 := #JOB_2_STEP_20)
      Contact( "Unit1.Em2.ControlNodes".jrOutPnPRight.sequence.status.seqActive )
      wire#w1
      Coil( "Unit1.Em2.ControlNodes".jrOutPnPRight."step".action1[220] )
   END_RUNG
   RUNG wire#w1
      Contact( "Unit1.EmNodes".emRelations.em03.sequence.topTapeFixStage.jobInterface.unloadJob5.clampRequest )
      wire#w2
      Coil( "Unit1.Em2.ControlNodes".jrOutPnPRight."step".transition1[220] )
   END_RUNG
   RUNG wire#w1
      Contact( "Unit1.Em2.ControlNodes".jrOutPnPRight."step".transition1[220] )
   END_RUNG wire#w2
   RUNG wire#w1
      Contact( "Unit1.Em2.ControlNodes".jrOutPnPRight."step".transition1[220] )
      { S7_Templates := "time_type := Time" } #statTonTime[220].TON(pt := T#500ms, et =>)
      Move(in := #JOB_2_STEP_21, out1 => "Unit1.Em2.ControlNodes".jrOutPnPRight.sequence.status.nextStep)
   END_RUNG
   // the same network as SCL:
   "Unit1.Em2.ControlNodes".jrOutPnPRight."step".action1[220] := ("Unit1.Em2.ControlNodes".jrOutPnPRight.sequence.status.currentStep = #JOB_2_STEP_20) AND "Unit1.Em2.ControlNodes".jrOutPnPRight.sequence.status.seqActive;
   "Unit1.Em2.ControlNodes".jrOutPnPRight."step".transition1[220] := ("Unit1.Em2.ControlNodes".jrOutPnPRight.sequence.status.currentStep = #JOB_2_STEP_20) AND "Unit1.Em2.ControlNodes".jrOutPnPRight.sequence.status.seqActive AND ("Unit1.EmNodes".emRelations.em03.sequence.topTapeFixStage.jobInterface.unloadJob5.clampRequest OR "Unit1.Em2.ControlNodes".jrOutPnPRight."step".transition1[220]);
   #statTonTime[220].TON(IN := ("Unit1.Em2.ControlNodes".jrOutPnPRight.sequence.status.currentStep = #JOB_2_STEP_20) AND "Unit1.Em2.ControlNodes".jrOutPnPRight.sequence.status.seqActive AND "Unit1.Em2.ControlNodes".jrOutPnPRight."step".transition1[220],
                         PT := T#500ms);
   IF #statTonTime[220].Q THEN
       "Unit1.Em2.ControlNodes".jrOutPnPRight.sequence.status.nextStep := #JOB_2_STEP_21;
   END_IF;
END_REGION

REGION Network 18: Step[221] : JR PP Right Clamp Close
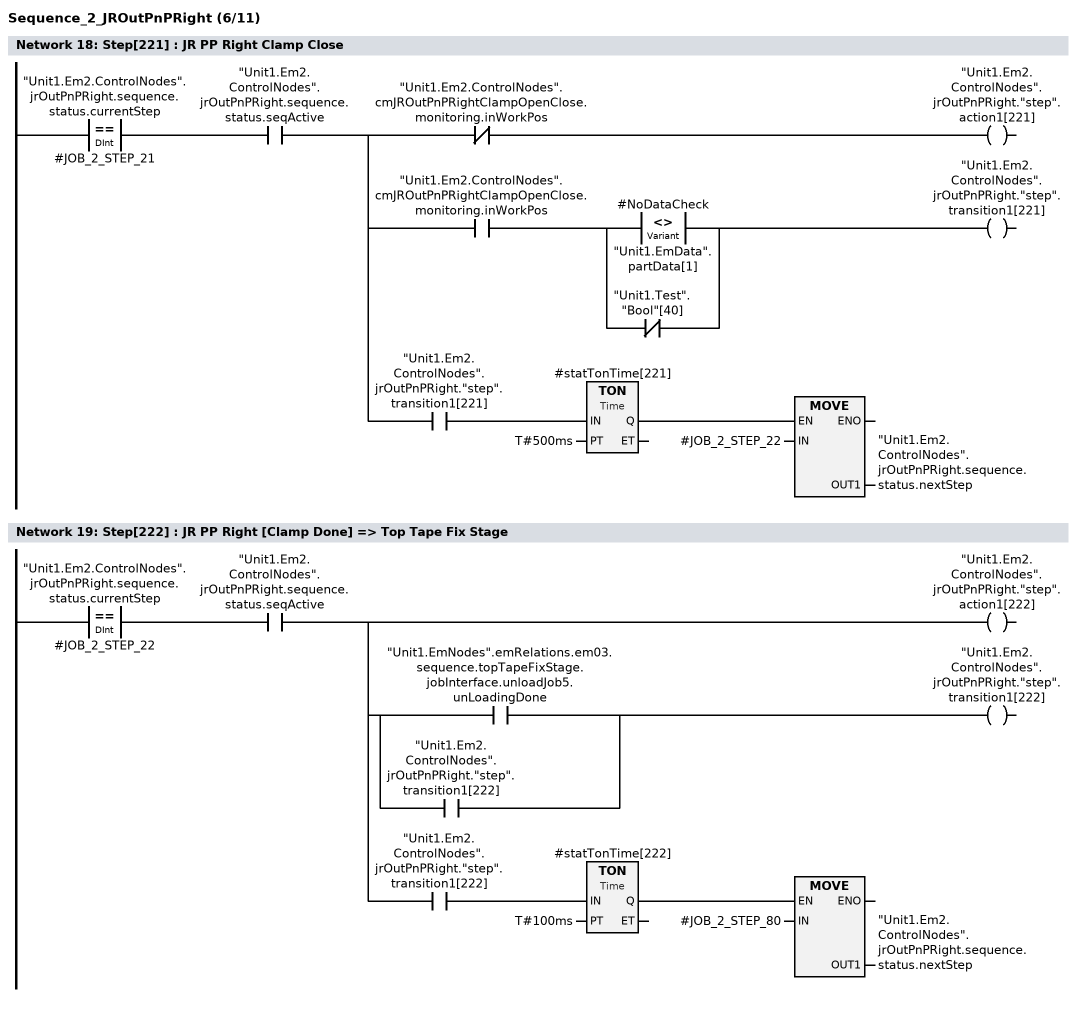
   RUNG wire#powerrail
      { S7_Templates := "SrcType := DInt" } EQ_Contact(in1 := "Unit1.Em2.ControlNodes".jrOutPnPRight.sequence.status.currentStep, in2 := #JOB_2_STEP_21)
      Contact( "Unit1.Em2.ControlNodes".jrOutPnPRight.sequence.status.seqActive )
      wire#w1
      I_Contact( "Unit1.Em2.ControlNodes".cmJROutPnPRightClampOpenClose.monitoring.inWorkPos )
      Coil( "Unit1.Em2.ControlNodes".jrOutPnPRight."step".action1[221] )
   END_RUNG
   RUNG wire#w1
      Contact( "Unit1.Em2.ControlNodes".cmJROutPnPRightClampOpenClose.monitoring.inWorkPos )
      wire#w2
      { S7_Templates := "SrcType := Variant" } NE_Contact(in1 := #NoDataCheck, in2 := "Unit1.EmData".partData[1])
      wire#w3
      Coil( "Unit1.Em2.ControlNodes".jrOutPnPRight."step".transition1[221] )
   END_RUNG
   RUNG wire#w2
      I_Contact( "Unit1.Test"."Bool"[40] )
   END_RUNG wire#w3
   RUNG wire#w1
      Contact( "Unit1.Em2.ControlNodes".jrOutPnPRight."step".transition1[221] )
      { S7_Templates := "time_type := Time" } #statTonTime[221].TON(pt := T#500ms, et =>)
      Move(in := #JOB_2_STEP_22, out1 => "Unit1.Em2.ControlNodes".jrOutPnPRight.sequence.status.nextStep)
   END_RUNG
   // the same network as SCL:
   #_w1 := ("Unit1.Em2.ControlNodes".jrOutPnPRight.sequence.status.currentStep = #JOB_2_STEP_21) AND "Unit1.Em2.ControlNodes".jrOutPnPRight.sequence.status.seqActive;
   "Unit1.Em2.ControlNodes".jrOutPnPRight."step".action1[221] := #_w1 AND NOT "Unit1.Em2.ControlNodes".cmJROutPnPRightClampOpenClose.monitoring.inWorkPos;
   "Unit1.Em2.ControlNodes".jrOutPnPRight."step".transition1[221] := #_w1 AND "Unit1.Em2.ControlNodes".cmJROutPnPRightClampOpenClose.monitoring.inWorkPos AND ((#NoDataCheck <> "Unit1.EmData".partData[1]) OR NOT "Unit1.Test"."Bool"[40]);
   #statTonTime[221].TON(IN := #_w1 AND "Unit1.Em2.ControlNodes".jrOutPnPRight."step".transition1[221],
                         PT := T#500ms);
   IF #statTonTime[221].Q THEN
       "Unit1.Em2.ControlNodes".jrOutPnPRight.sequence.status.nextStep := #JOB_2_STEP_22;
   END_IF;
END_REGION

REGION Network 19: Step[222] : JR PP Right [Clamp Done] => Top Tape Fix Stage
   RUNG wire#powerrail
      { S7_Templates := "SrcType := DInt" } EQ_Contact(in1 := "Unit1.Em2.ControlNodes".jrOutPnPRight.sequence.status.currentStep, in2 := #JOB_2_STEP_22)
      Contact( "Unit1.Em2.ControlNodes".jrOutPnPRight.sequence.status.seqActive )
      wire#w1
      Coil( "Unit1.Em2.ControlNodes".jrOutPnPRight."step".action1[222] )
   END_RUNG
   RUNG wire#w1
      Contact( "Unit1.EmNodes".emRelations.em03.sequence.topTapeFixStage.jobInterface.unloadJob5.unLoadingDone )
      wire#w2
      Coil( "Unit1.Em2.ControlNodes".jrOutPnPRight."step".transition1[222] )
   END_RUNG
   RUNG wire#w1
      Contact( "Unit1.Em2.ControlNodes".jrOutPnPRight."step".transition1[222] )
   END_RUNG wire#w2
   RUNG wire#w1
      Contact( "Unit1.Em2.ControlNodes".jrOutPnPRight."step".transition1[222] )
      { S7_Templates := "time_type := Time" } #statTonTime[222].TON(pt := T#100ms, et =>)
      Move(in := #JOB_2_STEP_80, out1 => "Unit1.Em2.ControlNodes".jrOutPnPRight.sequence.status.nextStep)
   END_RUNG
   // the same network as SCL:
   "Unit1.Em2.ControlNodes".jrOutPnPRight."step".action1[222] := ("Unit1.Em2.ControlNodes".jrOutPnPRight.sequence.status.currentStep = #JOB_2_STEP_22) AND "Unit1.Em2.ControlNodes".jrOutPnPRight.sequence.status.seqActive;
   "Unit1.Em2.ControlNodes".jrOutPnPRight."step".transition1[222] := ("Unit1.Em2.ControlNodes".jrOutPnPRight.sequence.status.currentStep = #JOB_2_STEP_22) AND "Unit1.Em2.ControlNodes".jrOutPnPRight.sequence.status.seqActive AND ("Unit1.EmNodes".emRelations.em03.sequence.topTapeFixStage.jobInterface.unloadJob5.unLoadingDone OR "Unit1.Em2.ControlNodes".jrOutPnPRight."step".transition1[222]);
   #statTonTime[222].TON(IN := ("Unit1.Em2.ControlNodes".jrOutPnPRight.sequence.status.currentStep = #JOB_2_STEP_22) AND "Unit1.Em2.ControlNodes".jrOutPnPRight.sequence.status.seqActive AND "Unit1.Em2.ControlNodes".jrOutPnPRight."step".transition1[222],
                         PT := T#100ms);
   IF #statTonTime[222].Q THEN
       "Unit1.Em2.ControlNodes".jrOutPnPRight.sequence.status.nextStep := #JOB_2_STEP_80;
   END_IF;
END_REGION

REGION Network 20: Step[280] : JR PP Right X/Z-Axis Wait Pos
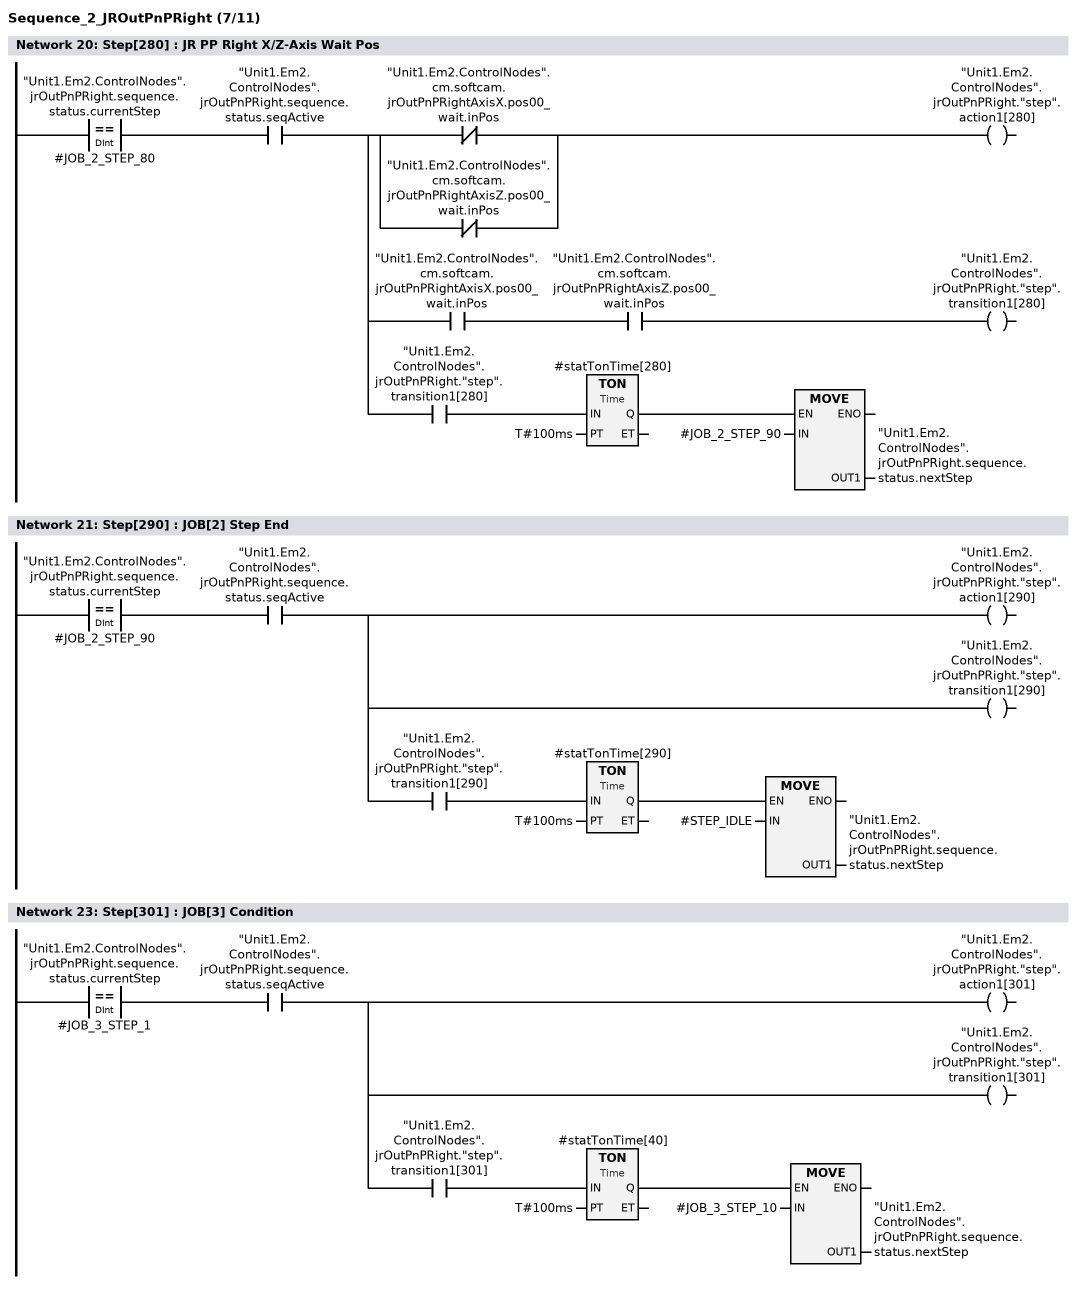
   RUNG wire#powerrail
      { S7_Templates := "SrcType := DInt" } EQ_Contact(in1 := "Unit1.Em2.ControlNodes".jrOutPnPRight.sequence.status.currentStep, in2 := #JOB_2_STEP_80)
      Contact( "Unit1.Em2.ControlNodes".jrOutPnPRight.sequence.status.seqActive )
      wire#w1
      I_Contact( "Unit1.Em2.ControlNodes".cm.softcam.jrOutPnPRightAxisX.pos00_wait.inPos )
      wire#w2
      Coil( "Unit1.Em2.ControlNodes".jrOutPnPRight."step".action1[280] )
   END_RUNG
   RUNG wire#w1
      I_Contact( "Unit1.Em2.ControlNodes".cm.softcam.jrOutPnPRightAxisZ.pos00_wait.inPos )
   END_RUNG wire#w2
   RUNG wire#w1
      Contact( "Unit1.Em2.ControlNodes".cm.softcam.jrOutPnPRightAxisX.pos00_wait.inPos )
      Contact( "Unit1.Em2.ControlNodes".cm.softcam.jrOutPnPRightAxisZ.pos00_wait.inPos )
      Coil( "Unit1.Em2.ControlNodes".jrOutPnPRight."step".transition1[280] )
   END_RUNG
   RUNG wire#w1
      Contact( "Unit1.Em2.ControlNodes".jrOutPnPRight."step".transition1[280] )
      { S7_Templates := "time_type := Time" } #statTonTime[280].TON(pt := T#100ms, et =>)
      Move(in := #JOB_2_STEP_90, out1 => "Unit1.Em2.ControlNodes".jrOutPnPRight.sequence.status.nextStep)
   END_RUNG
   // the same network as SCL:
   #_w1 := ("Unit1.Em2.ControlNodes".jrOutPnPRight.sequence.status.currentStep = #JOB_2_STEP_80) AND "Unit1.Em2.ControlNodes".jrOutPnPRight.sequence.status.seqActive;
   "Unit1.Em2.ControlNodes".jrOutPnPRight."step".action1[280] := #_w1 AND (NOT "Unit1.Em2.ControlNodes".cm.softcam.jrOutPnPRightAxisX.pos00_wait.inPos OR NOT "Unit1.Em2.ControlNodes".cm.softcam.jrOutPnPRightAxisZ.pos00_wait.inPos);
   "Unit1.Em2.ControlNodes".jrOutPnPRight."step".transition1[280] := #_w1 AND "Unit1.Em2.ControlNodes".cm.softcam.jrOutPnPRightAxisX.pos00_wait.inPos AND "Unit1.Em2.ControlNodes".cm.softcam.jrOutPnPRightAxisZ.pos00_wait.inPos;
   #statTonTime[280].TON(IN := #_w1 AND "Unit1.Em2.ControlNodes".jrOutPnPRight."step".transition1[280],
                         PT := T#100ms);
   IF #statTonTime[280].Q THEN
       "Unit1.Em2.ControlNodes".jrOutPnPRight.sequence.status.nextStep := #JOB_2_STEP_90;
   END_IF;
END_REGION

REGION Network 21: Step[290] : JOB[2] Step End
   RUNG wire#powerrail
      { S7_Templates := "SrcType := DInt" } EQ_Contact(in1 := "Unit1.Em2.ControlNodes".jrOutPnPRight.sequence.status.currentStep, in2 := #JOB_2_STEP_90)
      Contact( "Unit1.Em2.ControlNodes".jrOutPnPRight.sequence.status.seqActive )
      wire#w1
      Coil( "Unit1.Em2.ControlNodes".jrOutPnPRight."step".action1[290] )
   END_RUNG
   RUNG wire#w1
      Coil( "Unit1.Em2.ControlNodes".jrOutPnPRight."step".transition1[290] )
   END_RUNG
   RUNG wire#w1
      Contact( "Unit1.Em2.ControlNodes".jrOutPnPRight."step".transition1[290] )
      { S7_Templates := "time_type := Time" } #statTonTime[290].TON(pt := T#100ms, et =>)
      Move(in := #STEP_IDLE, out1 => "Unit1.Em2.ControlNodes".jrOutPnPRight.sequence.status.nextStep)
   END_RUNG
   // the same network as SCL:
   "Unit1.Em2.ControlNodes".jrOutPnPRight."step".action1[290] := ("Unit1.Em2.ControlNodes".jrOutPnPRight.sequence.status.currentStep = #JOB_2_STEP_90) AND "Unit1.Em2.ControlNodes".jrOutPnPRight.sequence.status.seqActive;
   "Unit1.Em2.ControlNodes".jrOutPnPRight."step".transition1[290] := ("Unit1.Em2.ControlNodes".jrOutPnPRight.sequence.status.currentStep = #JOB_2_STEP_90) AND "Unit1.Em2.ControlNodes".jrOutPnPRight.sequence.status.seqActive;
   #statTonTime[290].TON(IN := ("Unit1.Em2.ControlNodes".jrOutPnPRight.sequence.status.currentStep = #JOB_2_STEP_90) AND "Unit1.Em2.ControlNodes".jrOutPnPRight.sequence.status.seqActive AND "Unit1.Em2.ControlNodes".jrOutPnPRight."step".transition1[290],
                         PT := T#100ms);
   IF #statTonTime[290].Q THEN
       "Unit1.Em2.ControlNodes".jrOutPnPRight.sequence.status.nextStep := #STEP_IDLE;
   END_IF;
END_REGION

REGION Network 22: *************** JOB[3] JR PUT SIDE FIX STAGE=AUTO *************************
END_REGION

REGION Network 23: Step[301] : JOB[3] Condition
   RUNG wire#powerrail
      { S7_Templates := "SrcType := DInt" } EQ_Contact(in1 := "Unit1.Em2.ControlNodes".jrOutPnPRight.sequence.status.currentStep, in2 := #JOB_3_STEP_1)
      Contact( "Unit1.Em2.ControlNodes".jrOutPnPRight.sequence.status.seqActive )
      wire#w1
      Coil( "Unit1.Em2.ControlNodes".jrOutPnPRight."step".action1[301] )
   END_RUNG
   RUNG wire#w1
      Coil( "Unit1.Em2.ControlNodes".jrOutPnPRight."step".transition1[301] )
   END_RUNG
   RUNG wire#w1
      Contact( "Unit1.Em2.ControlNodes".jrOutPnPRight."step".transition1[301] )
      { S7_Templates := "time_type := Time" } #statTonTime[40].TON(pt := T#100ms, et =>)
      Move(in := #JOB_3_STEP_10, out1 => "Unit1.Em2.ControlNodes".jrOutPnPRight.sequence.status.nextStep)
   END_RUNG
   // the same network as SCL:
   "Unit1.Em2.ControlNodes".jrOutPnPRight."step".action1[301] := ("Unit1.Em2.ControlNodes".jrOutPnPRight.sequence.status.currentStep = #JOB_3_STEP_1) AND "Unit1.Em2.ControlNodes".jrOutPnPRight.sequence.status.seqActive;
   "Unit1.Em2.ControlNodes".jrOutPnPRight."step".transition1[301] := ("Unit1.Em2.ControlNodes".jrOutPnPRight.sequence.status.currentStep = #JOB_3_STEP_1) AND "Unit1.Em2.ControlNodes".jrOutPnPRight.sequence.status.seqActive;
   #statTonTime[40].TON(IN := ("Unit1.Em2.ControlNodes".jrOutPnPRight.sequence.status.currentStep = #JOB_3_STEP_1) AND "Unit1.Em2.ControlNodes".jrOutPnPRight.sequence.status.seqActive AND "Unit1.Em2.ControlNodes".jrOutPnPRight."step".transition1[301],
                        PT := T#100ms);
   IF #statTonTime[40].Q THEN
       "Unit1.Em2.ControlNodes".jrOutPnPRight.sequence.status.nextStep := #JOB_3_STEP_10;
   END_IF;
END_REGION

REGION Network 24: Step[310] : JR PP Right X-Axis Put Pos
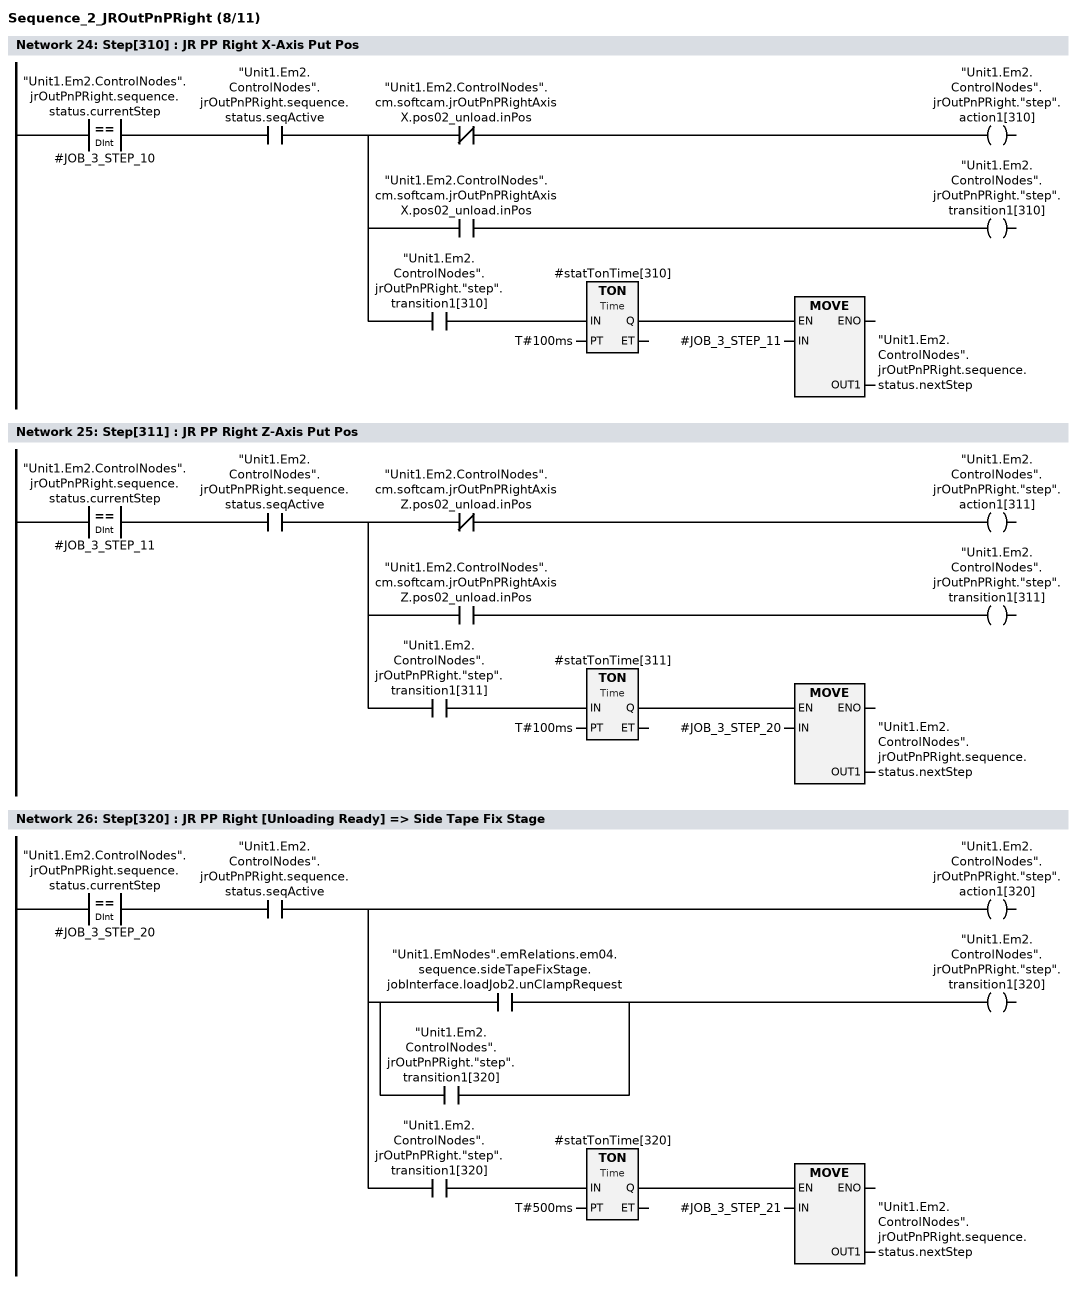
   RUNG wire#powerrail
      { S7_Templates := "SrcType := DInt" } EQ_Contact(in1 := "Unit1.Em2.ControlNodes".jrOutPnPRight.sequence.status.currentStep, in2 := #JOB_3_STEP_10)
      Contact( "Unit1.Em2.ControlNodes".jrOutPnPRight.sequence.status.seqActive )
      wire#w1
      I_Contact( "Unit1.Em2.ControlNodes".cm.softcam.jrOutPnPRightAxisX.pos02_unload.inPos )
      Coil( "Unit1.Em2.ControlNodes".jrOutPnPRight."step".action1[310] )
   END_RUNG
   RUNG wire#w1
      Contact( "Unit1.Em2.ControlNodes".cm.softcam.jrOutPnPRightAxisX.pos02_unload.inPos )
      Coil( "Unit1.Em2.ControlNodes".jrOutPnPRight."step".transition1[310] )
   END_RUNG
   RUNG wire#w1
      Contact( "Unit1.Em2.ControlNodes".jrOutPnPRight."step".transition1[310] )
      { S7_Templates := "time_type := Time" } #statTonTime[310].TON(pt := T#100ms, et =>)
      Move(in := #JOB_3_STEP_11, out1 => "Unit1.Em2.ControlNodes".jrOutPnPRight.sequence.status.nextStep)
   END_RUNG
   // the same network as SCL:
   #_w1 := ("Unit1.Em2.ControlNodes".jrOutPnPRight.sequence.status.currentStep = #JOB_3_STEP_10) AND "Unit1.Em2.ControlNodes".jrOutPnPRight.sequence.status.seqActive;
   "Unit1.Em2.ControlNodes".jrOutPnPRight."step".action1[310] := #_w1 AND NOT "Unit1.Em2.ControlNodes".cm.softcam.jrOutPnPRightAxisX.pos02_unload.inPos;
   "Unit1.Em2.ControlNodes".jrOutPnPRight."step".transition1[310] := #_w1 AND "Unit1.Em2.ControlNodes".cm.softcam.jrOutPnPRightAxisX.pos02_unload.inPos;
   #statTonTime[310].TON(IN := #_w1 AND "Unit1.Em2.ControlNodes".jrOutPnPRight."step".transition1[310],
                         PT := T#100ms);
   IF #statTonTime[310].Q THEN
       "Unit1.Em2.ControlNodes".jrOutPnPRight.sequence.status.nextStep := #JOB_3_STEP_11;
   END_IF;
END_REGION

REGION Network 25: Step[311] : JR PP Right Z-Axis Put Pos
   RUNG wire#powerrail
      { S7_Templates := "SrcType := DInt" } EQ_Contact(in1 := "Unit1.Em2.ControlNodes".jrOutPnPRight.sequence.status.currentStep, in2 := #JOB_3_STEP_11)
      Contact( "Unit1.Em2.ControlNodes".jrOutPnPRight.sequence.status.seqActive )
      wire#w1
      I_Contact( "Unit1.Em2.ControlNodes".cm.softcam.jrOutPnPRightAxisZ.pos02_unload.inPos )
      Coil( "Unit1.Em2.ControlNodes".jrOutPnPRight."step".action1[311] )
   END_RUNG
   RUNG wire#w1
      Contact( "Unit1.Em2.ControlNodes".cm.softcam.jrOutPnPRightAxisZ.pos02_unload.inPos )
      Coil( "Unit1.Em2.ControlNodes".jrOutPnPRight."step".transition1[311] )
   END_RUNG
   RUNG wire#w1
      Contact( "Unit1.Em2.ControlNodes".jrOutPnPRight."step".transition1[311] )
      { S7_Templates := "time_type := Time" } #statTonTime[311].TON(pt := T#100ms, et =>)
      Move(in := #JOB_3_STEP_20, out1 => "Unit1.Em2.ControlNodes".jrOutPnPRight.sequence.status.nextStep)
   END_RUNG
   // the same network as SCL:
   #_w1 := ("Unit1.Em2.ControlNodes".jrOutPnPRight.sequence.status.currentStep = #JOB_3_STEP_11) AND "Unit1.Em2.ControlNodes".jrOutPnPRight.sequence.status.seqActive;
   "Unit1.Em2.ControlNodes".jrOutPnPRight."step".action1[311] := #_w1 AND NOT "Unit1.Em2.ControlNodes".cm.softcam.jrOutPnPRightAxisZ.pos02_unload.inPos;
   "Unit1.Em2.ControlNodes".jrOutPnPRight."step".transition1[311] := #_w1 AND "Unit1.Em2.ControlNodes".cm.softcam.jrOutPnPRightAxisZ.pos02_unload.inPos;
   #statTonTime[311].TON(IN := #_w1 AND "Unit1.Em2.ControlNodes".jrOutPnPRight."step".transition1[311],
                         PT := T#100ms);
   IF #statTonTime[311].Q THEN
       "Unit1.Em2.ControlNodes".jrOutPnPRight.sequence.status.nextStep := #JOB_3_STEP_20;
   END_IF;
END_REGION

REGION Network 26: Step[320] : JR PP Right [Unloading Ready] => Side Tape Fix Stage
   RUNG wire#powerrail
      { S7_Templates := "SrcType := DInt" } EQ_Contact(in1 := "Unit1.Em2.ControlNodes".jrOutPnPRight.sequence.status.currentStep, in2 := #JOB_3_STEP_20)
      Contact( "Unit1.Em2.ControlNodes".jrOutPnPRight.sequence.status.seqActive )
      wire#w1
      Coil( "Unit1.Em2.ControlNodes".jrOutPnPRight."step".action1[320] )
   END_RUNG
   RUNG wire#w1
      Contact( "Unit1.EmNodes".emRelations.em04.sequence.sideTapeFixStage.jobInterface.loadJob2.unClampRequest )
      wire#w2
      Coil( "Unit1.Em2.ControlNodes".jrOutPnPRight."step".transition1[320] )
   END_RUNG
   RUNG wire#w1
      Contact( "Unit1.Em2.ControlNodes".jrOutPnPRight."step".transition1[320] )
   END_RUNG wire#w2
   RUNG wire#w1
      Contact( "Unit1.Em2.ControlNodes".jrOutPnPRight."step".transition1[320] )
      { S7_Templates := "time_type := Time" } #statTonTime[320].TON(pt := T#500ms, et =>)
      Move(in := #JOB_3_STEP_21, out1 => "Unit1.Em2.ControlNodes".jrOutPnPRight.sequence.status.nextStep)
   END_RUNG
   // the same network as SCL:
   "Unit1.Em2.ControlNodes".jrOutPnPRight."step".action1[320] := ("Unit1.Em2.ControlNodes".jrOutPnPRight.sequence.status.currentStep = #JOB_3_STEP_20) AND "Unit1.Em2.ControlNodes".jrOutPnPRight.sequence.status.seqActive;
   "Unit1.Em2.ControlNodes".jrOutPnPRight."step".transition1[320] := ("Unit1.Em2.ControlNodes".jrOutPnPRight.sequence.status.currentStep = #JOB_3_STEP_20) AND "Unit1.Em2.ControlNodes".jrOutPnPRight.sequence.status.seqActive AND ("Unit1.EmNodes".emRelations.em04.sequence.sideTapeFixStage.jobInterface.loadJob2.unClampRequest OR "Unit1.Em2.ControlNodes".jrOutPnPRight."step".transition1[320]);
   #statTonTime[320].TON(IN := ("Unit1.Em2.ControlNodes".jrOutPnPRight.sequence.status.currentStep = #JOB_3_STEP_20) AND "Unit1.Em2.ControlNodes".jrOutPnPRight.sequence.status.seqActive AND "Unit1.Em2.ControlNodes".jrOutPnPRight."step".transition1[320],
                         PT := T#500ms);
   IF #statTonTime[320].Q THEN
       "Unit1.Em2.ControlNodes".jrOutPnPRight.sequence.status.nextStep := #JOB_3_STEP_21;
   END_IF;
END_REGION

REGION Network 27: Step[321] : JR PP Right Clamp Open
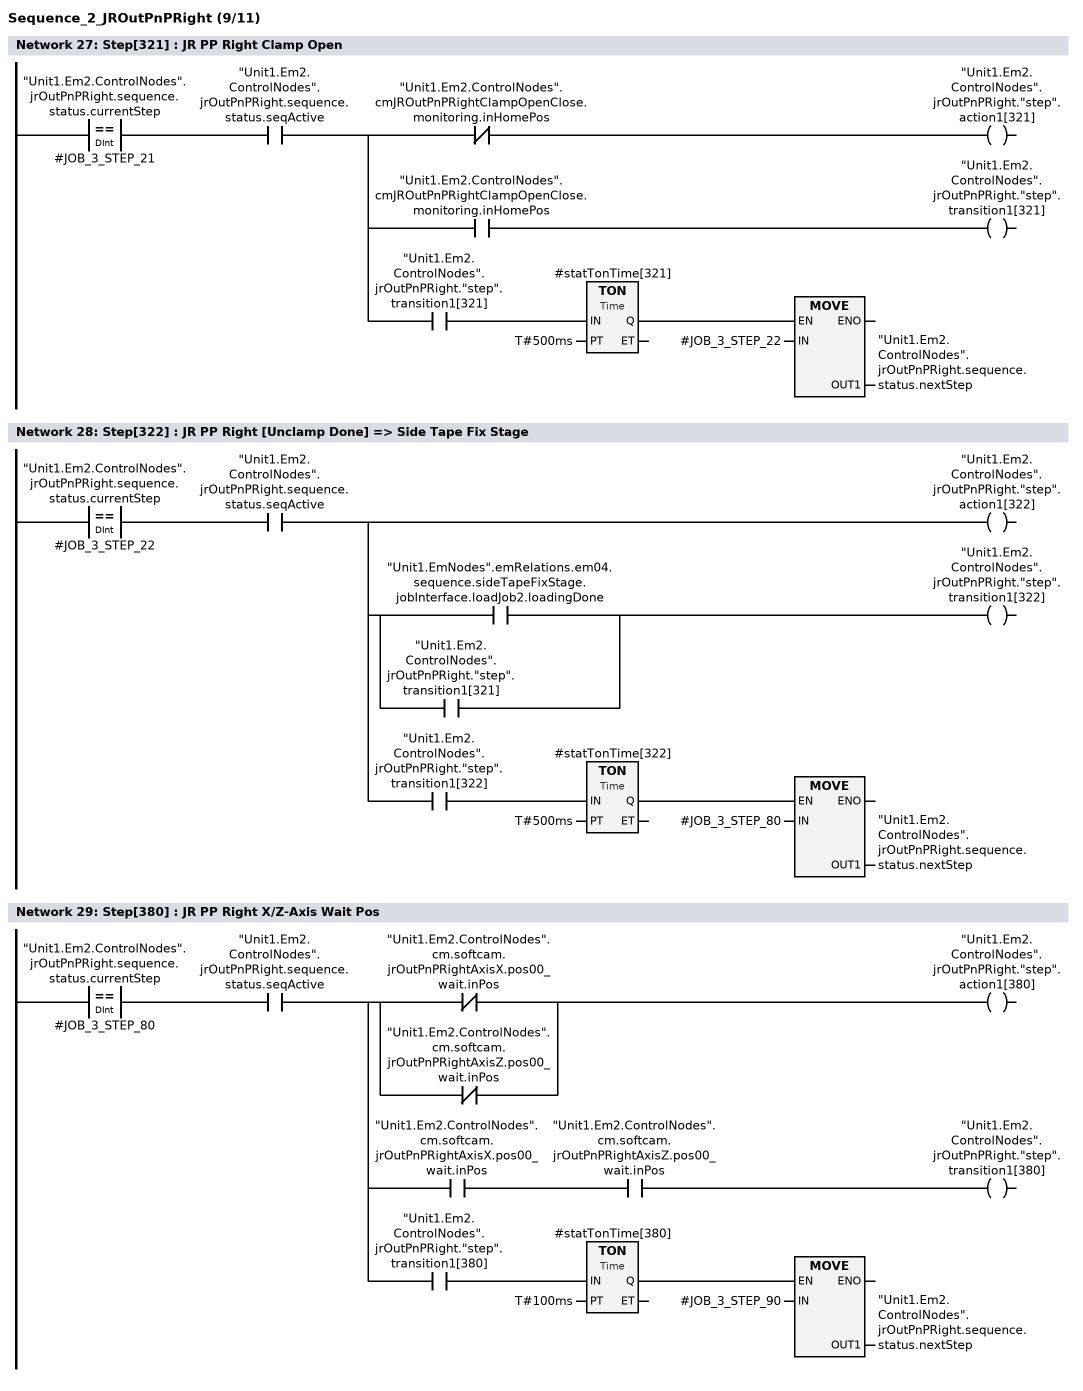
   RUNG wire#powerrail
      { S7_Templates := "SrcType := DInt" } EQ_Contact(in1 := "Unit1.Em2.ControlNodes".jrOutPnPRight.sequence.status.currentStep, in2 := #JOB_3_STEP_21)
      Contact( "Unit1.Em2.ControlNodes".jrOutPnPRight.sequence.status.seqActive )
      wire#w1
      I_Contact( "Unit1.Em2.ControlNodes".cmJROutPnPRightClampOpenClose.monitoring.inHomePos )
      Coil( "Unit1.Em2.ControlNodes".jrOutPnPRight."step".action1[321] )
   END_RUNG
   RUNG wire#w1
      Contact( "Unit1.Em2.ControlNodes".cmJROutPnPRightClampOpenClose.monitoring.inHomePos )
      Coil( "Unit1.Em2.ControlNodes".jrOutPnPRight."step".transition1[321] )
   END_RUNG
   RUNG wire#w1
      Contact( "Unit1.Em2.ControlNodes".jrOutPnPRight."step".transition1[321] )
      { S7_Templates := "time_type := Time" } #statTonTime[321].TON(pt := T#500ms, et =>)
      Move(in := #JOB_3_STEP_22, out1 => "Unit1.Em2.ControlNodes".jrOutPnPRight.sequence.status.nextStep)
   END_RUNG
   // the same network as SCL:
   #_w1 := ("Unit1.Em2.ControlNodes".jrOutPnPRight.sequence.status.currentStep = #JOB_3_STEP_21) AND "Unit1.Em2.ControlNodes".jrOutPnPRight.sequence.status.seqActive;
   "Unit1.Em2.ControlNodes".jrOutPnPRight."step".action1[321] := #_w1 AND NOT "Unit1.Em2.ControlNodes".cmJROutPnPRightClampOpenClose.monitoring.inHomePos;
   "Unit1.Em2.ControlNodes".jrOutPnPRight."step".transition1[321] := #_w1 AND "Unit1.Em2.ControlNodes".cmJROutPnPRightClampOpenClose.monitoring.inHomePos;
   #statTonTime[321].TON(IN := #_w1 AND "Unit1.Em2.ControlNodes".jrOutPnPRight."step".transition1[321],
                         PT := T#500ms);
   IF #statTonTime[321].Q THEN
       "Unit1.Em2.ControlNodes".jrOutPnPRight.sequence.status.nextStep := #JOB_3_STEP_22;
   END_IF;
END_REGION

REGION Network 28: Step[322] : JR PP Right [Unclamp Done] => Side Tape Fix Stage
   RUNG wire#powerrail
      { S7_Templates := "SrcType := DInt" } EQ_Contact(in1 := "Unit1.Em2.ControlNodes".jrOutPnPRight.sequence.status.currentStep, in2 := #JOB_3_STEP_22)
      Contact( "Unit1.Em2.ControlNodes".jrOutPnPRight.sequence.status.seqActive )
      wire#w1
      Coil( "Unit1.Em2.ControlNodes".jrOutPnPRight."step".action1[322] )
   END_RUNG
   RUNG wire#w1
      Contact( "Unit1.EmNodes".emRelations.em04.sequence.sideTapeFixStage.jobInterface.loadJob2.loadingDone )
      wire#w2
      Coil( "Unit1.Em2.ControlNodes".jrOutPnPRight."step".transition1[322] )
   END_RUNG
   RUNG wire#w1
      Contact( "Unit1.Em2.ControlNodes".jrOutPnPRight."step".transition1[321] )
   END_RUNG wire#w2
   RUNG wire#w1
      Contact( "Unit1.Em2.ControlNodes".jrOutPnPRight."step".transition1[322] )
      { S7_Templates := "time_type := Time" } #statTonTime[322].TON(pt := T#500ms, et =>)
      Move(in := #JOB_3_STEP_80, out1 => "Unit1.Em2.ControlNodes".jrOutPnPRight.sequence.status.nextStep)
   END_RUNG
   // the same network as SCL:
   "Unit1.Em2.ControlNodes".jrOutPnPRight."step".action1[322] := ("Unit1.Em2.ControlNodes".jrOutPnPRight.sequence.status.currentStep = #JOB_3_STEP_22) AND "Unit1.Em2.ControlNodes".jrOutPnPRight.sequence.status.seqActive;
   "Unit1.Em2.ControlNodes".jrOutPnPRight."step".transition1[322] := ("Unit1.Em2.ControlNodes".jrOutPnPRight.sequence.status.currentStep = #JOB_3_STEP_22) AND "Unit1.Em2.ControlNodes".jrOutPnPRight.sequence.status.seqActive AND ("Unit1.EmNodes".emRelations.em04.sequence.sideTapeFixStage.jobInterface.loadJob2.loadingDone OR "Unit1.Em2.ControlNodes".jrOutPnPRight."step".transition1[321]);
   #statTonTime[322].TON(IN := ("Unit1.Em2.ControlNodes".jrOutPnPRight.sequence.status.currentStep = #JOB_3_STEP_22) AND "Unit1.Em2.ControlNodes".jrOutPnPRight.sequence.status.seqActive AND "Unit1.Em2.ControlNodes".jrOutPnPRight."step".transition1[322],
                         PT := T#500ms);
   IF #statTonTime[322].Q THEN
       "Unit1.Em2.ControlNodes".jrOutPnPRight.sequence.status.nextStep := #JOB_3_STEP_80;
   END_IF;
END_REGION

REGION Network 29: Step[380] : JR PP Right X/Z-Axis Wait Pos
   RUNG wire#powerrail
      { S7_Templates := "SrcType := DInt" } EQ_Contact(in1 := "Unit1.Em2.ControlNodes".jrOutPnPRight.sequence.status.currentStep, in2 := #JOB_3_STEP_80)
      Contact( "Unit1.Em2.ControlNodes".jrOutPnPRight.sequence.status.seqActive )
      wire#w1
      I_Contact( "Unit1.Em2.ControlNodes".cm.softcam.jrOutPnPRightAxisX.pos00_wait.inPos )
      wire#w2
      Coil( "Unit1.Em2.ControlNodes".jrOutPnPRight."step".action1[380] )
   END_RUNG
   RUNG wire#w1
      I_Contact( "Unit1.Em2.ControlNodes".cm.softcam.jrOutPnPRightAxisZ.pos00_wait.inPos )
   END_RUNG wire#w2
   RUNG wire#w1
      Contact( "Unit1.Em2.ControlNodes".cm.softcam.jrOutPnPRightAxisX.pos00_wait.inPos )
      Contact( "Unit1.Em2.ControlNodes".cm.softcam.jrOutPnPRightAxisZ.pos00_wait.inPos )
      Coil( "Unit1.Em2.ControlNodes".jrOutPnPRight."step".transition1[380] )
   END_RUNG
   RUNG wire#w1
      Contact( "Unit1.Em2.ControlNodes".jrOutPnPRight."step".transition1[380] )
      { S7_Templates := "time_type := Time" } #statTonTime[380].TON(pt := T#100ms, et =>)
      Move(in := #JOB_3_STEP_90, out1 => "Unit1.Em2.ControlNodes".jrOutPnPRight.sequence.status.nextStep)
   END_RUNG
   // the same network as SCL:
   #_w1 := ("Unit1.Em2.ControlNodes".jrOutPnPRight.sequence.status.currentStep = #JOB_3_STEP_80) AND "Unit1.Em2.ControlNodes".jrOutPnPRight.sequence.status.seqActive;
   "Unit1.Em2.ControlNodes".jrOutPnPRight."step".action1[380] := #_w1 AND (NOT "Unit1.Em2.ControlNodes".cm.softcam.jrOutPnPRightAxisX.pos00_wait.inPos OR NOT "Unit1.Em2.ControlNodes".cm.softcam.jrOutPnPRightAxisZ.pos00_wait.inPos);
   "Unit1.Em2.ControlNodes".jrOutPnPRight."step".transition1[380] := #_w1 AND "Unit1.Em2.ControlNodes".cm.softcam.jrOutPnPRightAxisX.pos00_wait.inPos AND "Unit1.Em2.ControlNodes".cm.softcam.jrOutPnPRightAxisZ.pos00_wait.inPos;
   #statTonTime[380].TON(IN := #_w1 AND "Unit1.Em2.ControlNodes".jrOutPnPRight."step".transition1[380],
                         PT := T#100ms);
   IF #statTonTime[380].Q THEN
       "Unit1.Em2.ControlNodes".jrOutPnPRight.sequence.status.nextStep := #JOB_3_STEP_90;
   END_IF;
END_REGION

REGION Network 30: Step[390] : JOB[3] Step End
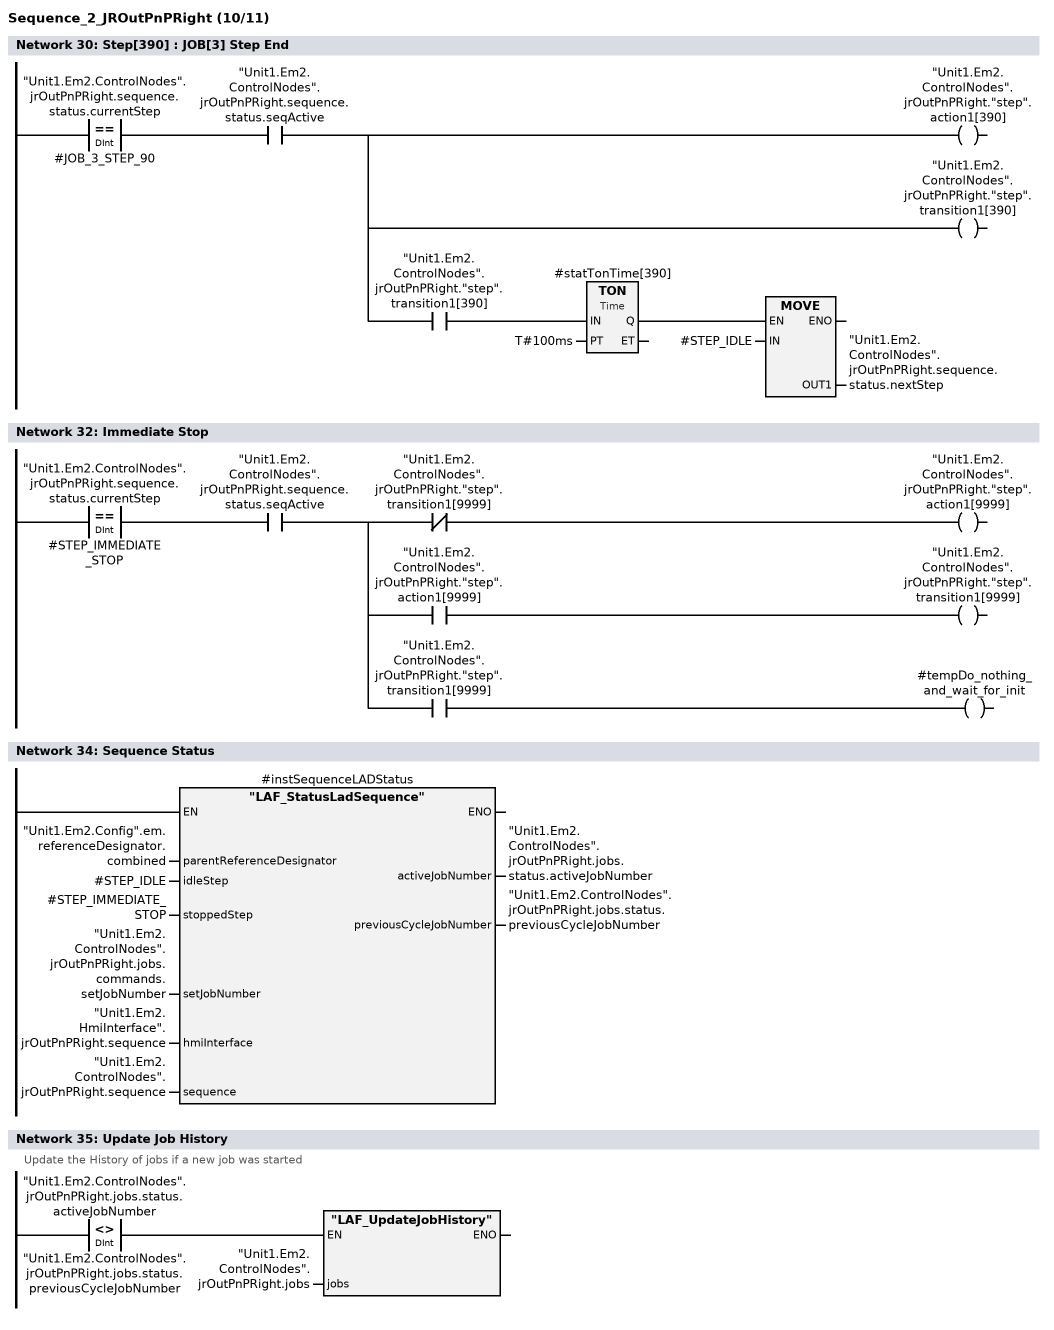
   RUNG wire#powerrail
      { S7_Templates := "SrcType := DInt" } EQ_Contact(in1 := "Unit1.Em2.ControlNodes".jrOutPnPRight.sequence.status.currentStep, in2 := #JOB_3_STEP_90)
      Contact( "Unit1.Em2.ControlNodes".jrOutPnPRight.sequence.status.seqActive )
      wire#w1
      Coil( "Unit1.Em2.ControlNodes".jrOutPnPRight."step".action1[390] )
   END_RUNG
   RUNG wire#w1
      Coil( "Unit1.Em2.ControlNodes".jrOutPnPRight."step".transition1[390] )
   END_RUNG
   RUNG wire#w1
      Contact( "Unit1.Em2.ControlNodes".jrOutPnPRight."step".transition1[390] )
      { S7_Templates := "time_type := Time" } #statTonTime[390].TON(pt := T#100ms, et =>)
      Move(in := #STEP_IDLE, out1 => "Unit1.Em2.ControlNodes".jrOutPnPRight.sequence.status.nextStep)
   END_RUNG
   // the same network as SCL:
   "Unit1.Em2.ControlNodes".jrOutPnPRight."step".action1[390] := ("Unit1.Em2.ControlNodes".jrOutPnPRight.sequence.status.currentStep = #JOB_3_STEP_90) AND "Unit1.Em2.ControlNodes".jrOutPnPRight.sequence.status.seqActive;
   "Unit1.Em2.ControlNodes".jrOutPnPRight."step".transition1[390] := ("Unit1.Em2.ControlNodes".jrOutPnPRight.sequence.status.currentStep = #JOB_3_STEP_90) AND "Unit1.Em2.ControlNodes".jrOutPnPRight.sequence.status.seqActive;
   #statTonTime[390].TON(IN := ("Unit1.Em2.ControlNodes".jrOutPnPRight.sequence.status.currentStep = #JOB_3_STEP_90) AND "Unit1.Em2.ControlNodes".jrOutPnPRight.sequence.status.seqActive AND "Unit1.Em2.ControlNodes".jrOutPnPRight."step".transition1[390],
                         PT := T#100ms);
   IF #statTonTime[390].Q THEN
       "Unit1.Em2.ControlNodes".jrOutPnPRight.sequence.status.nextStep := #STEP_IDLE;
   END_IF;
END_REGION

REGION Network 31: *************** IMMEDIATE STOP ****************
END_REGION

REGION Network 32: Immediate Stop
   RUNG wire#powerrail
      { S7_Templates := "SrcType := DInt" } EQ_Contact(in1 := "Unit1.Em2.ControlNodes".jrOutPnPRight.sequence.status.currentStep, in2 := #STEP_IMMEDIATE_STOP)
      Contact( "Unit1.Em2.ControlNodes".jrOutPnPRight.sequence.status.seqActive )
      wire#w1
      I_Contact( "Unit1.Em2.ControlNodes".jrOutPnPRight."step".transition1[9999] )
      Coil( "Unit1.Em2.ControlNodes".jrOutPnPRight."step".action1[9999] )
   END_RUNG
   RUNG wire#w1
      Contact( "Unit1.Em2.ControlNodes".jrOutPnPRight."step".action1[9999] )
      Coil( "Unit1.Em2.ControlNodes".jrOutPnPRight."step".transition1[9999] )
   END_RUNG
   RUNG wire#w1
      Contact( "Unit1.Em2.ControlNodes".jrOutPnPRight."step".transition1[9999] )
      Coil( #tempDo_nothing_and_wait_for_init )
   END_RUNG
   // the same network as SCL:
   #_w1 := ("Unit1.Em2.ControlNodes".jrOutPnPRight.sequence.status.currentStep = #STEP_IMMEDIATE_STOP) AND "Unit1.Em2.ControlNodes".jrOutPnPRight.sequence.status.seqActive;
   "Unit1.Em2.ControlNodes".jrOutPnPRight."step".action1[9999] := #_w1 AND NOT "Unit1.Em2.ControlNodes".jrOutPnPRight."step".transition1[9999];
   "Unit1.Em2.ControlNodes".jrOutPnPRight."step".transition1[9999] := #_w1 AND "Unit1.Em2.ControlNodes".jrOutPnPRight."step".action1[9999];
   #tempDo_nothing_and_wait_for_init := #_w1 AND "Unit1.Em2.ControlNodes".jrOutPnPRight."step".transition1[9999];
END_REGION

REGION Network 33: *************** STATUS **********************
END_REGION

REGION Network 34: Sequence Status
   RUNG wire#powerrail
      #instSequenceLADStatus(parentReferenceDesignator := "Unit1.Em2.Config".em.referenceDesignator.combined, idleStep := #STEP_IDLE, stoppedStep := #STEP_IMMEDIATE_STOP, setJobNumber := "Unit1.Em2.ControlNodes".jrOutPnPRight.jobs.commands.setJobNumber, hmiInterface := "Unit1.Em2.HmiInterface".jrOutPnPRight.sequence, sequence := "Unit1.Em2.ControlNodes".jrOutPnPRight.sequence, activeJobNumber => "Unit1.Em2.ControlNodes".jrOutPnPRight.jobs.status.activeJobNumber, previousCycleJobNumber => "Unit1.Em2.ControlNodes".jrOutPnPRight.jobs.status.previousCycleJobNumber)
   END_RUNG
   // the same network as SCL:
   #instSequenceLADStatus(parentReferenceDesignator := "Unit1.Em2.Config".em.referenceDesignator.combined,   // "LAF_StatusLadSequence"
                          idleStep := #STEP_IDLE,
                          stoppedStep := #STEP_IMMEDIATE_STOP,
                          setJobNumber := "Unit1.Em2.ControlNodes".jrOutPnPRight.jobs.commands.setJobNumber,
                          hmiInterface := "Unit1.Em2.HmiInterface".jrOutPnPRight.sequence,
                          sequence := "Unit1.Em2.ControlNodes".jrOutPnPRight.sequence,
                          activeJobNumber => "Unit1.Em2.ControlNodes".jrOutPnPRight.jobs.status.activeJobNumber,
                          previousCycleJobNumber => "Unit1.Em2.ControlNodes".jrOutPnPRight.jobs.status.previousCycleJobNumber);
END_REGION

REGION Network 35: Update Job History
   // Update the History of jobs if a new job was started
   RUNG wire#powerrail
      { S7_Templates := "SrcType := DInt" } NE_Contact(in1 := "Unit1.Em2.ControlNodes".jrOutPnPRight.jobs.status.activeJobNumber, in2 := "Unit1.Em2.ControlNodes".jrOutPnPRight.jobs.status.previousCycleJobNumber)
      "LAF_UpdateJobHistory"(jobs := "Unit1.Em2.ControlNodes".jrOutPnPRight.jobs)
   END_RUNG
   // the same network as SCL:
   IF "Unit1.Em2.ControlNodes".jrOutPnPRight.jobs.status.activeJobNumber <> "Unit1.Em2.ControlNodes".jrOutPnPRight.jobs.status.previousCycleJobNumber THEN
       "LAF_UpdateJobHistory"(jobs := "Unit1.Em2.ControlNodes".jrOutPnPRight.jobs);
   END_IF;
END_REGION

REGION Network 36: Output Steps As String
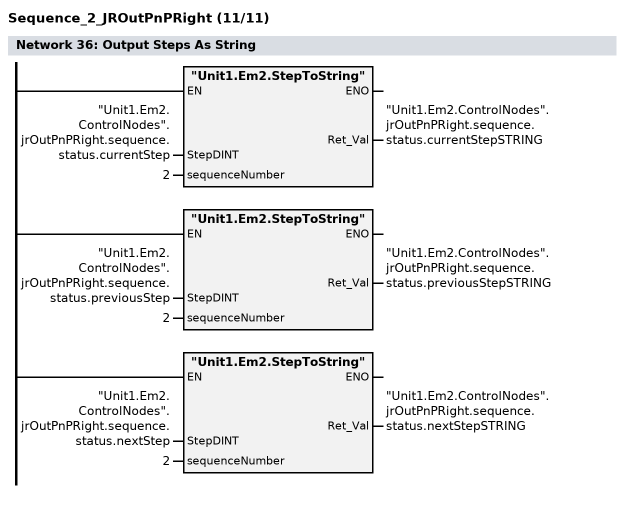
   RUNG wire#powerrail
      "Unit1.Em2.StepToString"(StepDINT := "Unit1.Em2.ControlNodes".jrOutPnPRight.sequence.status.currentStep, sequenceNumber := 2, Ret_Val => "Unit1.Em2.ControlNodes".jrOutPnPRight.sequence.status.currentStepSTRING)
   END_RUNG
   RUNG wire#powerrail
      "Unit1.Em2.StepToString"(StepDINT := "Unit1.Em2.ControlNodes".jrOutPnPRight.sequence.status.previousStep, sequenceNumber := 2, Ret_Val => "Unit1.Em2.ControlNodes".jrOutPnPRight.sequence.status.previousStepSTRING)
   END_RUNG
   RUNG wire#powerrail
      "Unit1.Em2.StepToString"(StepDINT := "Unit1.Em2.ControlNodes".jrOutPnPRight.sequence.status.nextStep, sequenceNumber := 2, Ret_Val => "Unit1.Em2.ControlNodes".jrOutPnPRight.sequence.status.nextStepSTRING)
   END_RUNG
   // the same network as SCL:
   "Unit1.Em2.ControlNodes".jrOutPnPRight.sequence.status.currentStepSTRING := "Unit1.Em2.StepToString"(StepDINT := "Unit1.Em2.ControlNodes".jrOutPnPRight.sequence.status.currentStep,
                           sequenceNumber := 2);
   "Unit1.Em2.ControlNodes".jrOutPnPRight.sequence.status.previousStepSTRING := "Unit1.Em2.StepToString"(StepDINT := "Unit1.Em2.ControlNodes".jrOutPnPRight.sequence.status.previousStep,
                           sequenceNumber := 2);
   "Unit1.Em2.ControlNodes".jrOutPnPRight.sequence.status.nextStepSTRING := "Unit1.Em2.StepToString"(StepDINT := "Unit1.Em2.ControlNodes".jrOutPnPRight.sequence.status.nextStep,
                           sequenceNumber := 2);
END_REGION
END_FUNCTION_BLOCK
